METHOD M_SetSingleProp : ERRORID
VAR_INPUT
	refCmdData : REFERENCE TO  ST_CmdData;
END_VAR
IF nSpecPropIndex = refCmdData.aHeader[1] THEN
	IF refCmdData.n32Data[0] > 0 AND refCmdData.n32Data[0] <= cNoOfValves THEN
		nValveNrVac := DINT_TO_USINT(refCmdData.n32Data[0]);
	ELSE
		M_SetSingleProp := E_ErrorIdObjMgmt.ERRORID_InvalidValveNumber;
	END_IF	
ELSE
	M_SetSingleProp := SUPER^.M_SetSingleProp(refCmdData);
END_IF
END_METHOD

END_FUNCTION_BLOCK

// ---- Hardware/HuberUnistat/FB_UnistatControl.TcPOU
FUNCTION_BLOCK FB_UnistatControl
VAR_INPUT
	UnistatRef 		: REFERENCE TO FB_HwRefUnistat;
	nTempSetpoint 	: DINT;
	bTempControlOn	: BOOL;
	bExecute		: BOOL;
END_VAR
VAR_OUTPUT
	bBusy			: BOOL;
	bError			: BOOL;
	nErrorID		: ERRORID;
END_VAR
VAR
	fbSendCmd 		: FB_Unistat_SendCmd;
	nState			: UINT;
END_VAR

IF bExecute THEN
	IF NOT __ISVALIDREF(UnistatRef) THEN
		{warnig 'Implement proper ErrorID'}
		bError := TRUE;
		nErrorID := 333;
		RETURN;
	END_IF
	fbSendCmd.SerialPort REF= UnistatRef.P_SerialPort;
 	UnistatRef.P_bPolling := FALSE;
	
	IF nState = 0 THEN
		IF UnistatRef.P_eState = E_UnistatState.Error THEN
			RETURN;
		END_IF
		IF bTempControlOn THEN
			IF UnistatRef.P_eState = E_UnistatState.On THEN
				nState := 3;
			ELSE
				nState := 1;
			END_IF
		ELSE
			IF UnistatRef.P_eState = E_UnistatState.On THEN
				nState := 2;
			ELSE
				RETURN;
			END_IF
		END_IF
		bBusy := TRUE;
	END_IF
	
	CASE nState OF
		1:	//Ein
			fbSendCmd(bExecute:= TRUE, eCommand:= E_Unitstat_Command.Start_TempControl);
			IF NOT fbSendCmd.bBusy THEN
				fbSendCmd(bExecute:= FALSE);
				nState := 3;
			END_IF
		
		2:	//Aus
			fbSendCmd(bExecute:= TRUE, eCommand:= E_Unitstat_Command.Stop_TempControl);
			IF NOT fbSendCmd.bBusy THEN
				fbSendCmd(bExecute:= FALSE);
				bBusy := FALSE;
				nState := 80;
			END_IF
		
		3:	//Solltemperatur
			fbSendCmd(bExecute:= TRUE, eCommand:= E_Unitstat_Command.Set_TempSetPoint, nSendData := nTempSetPoint);
			IF NOT fbSendCmd.bBusy THEN
				fbSendCmd(bExecute:= FALSE);
				bBusy := FALSE;
				nState := 80;
			END_IF
	END_CASE
ELSE
	IF __ISVALIDREF(UnistatRef) THEN
		UnistatRef.P_bPolling := TRUE;
	END_IF
	nState := 0;
	bBusy := FALSE;
	bError := FALSE;
	nErrorID := 0;
END_IF

END_FUNCTION_BLOCK

// ---- Hardware/HuberUnistat/FB_HwRefUnistat.TcPOU
FUNCTION_BLOCK FB_HwRefUnistat
VAR_INPUT
END_VAR
VAR_OUTPUT
END_VAR
VAR
	SerialPort 	: REFERENCE TO FB_SerialComPort_Base;
	fbSendCmd 	: FB_Unistat_SendCmd;
	
	bPolling			: BOOL := TRUE;
	nCurrentTempIntern 	: DINT;
	nCurrentTempExtern 	: DINT;
	eState				: E_UnistatState;
	nState				: USINT;
	nStateNext			: USINT := 1;
END_VAR

IF NOT __ISVALIDREF(SerialPort) THEN
	RETURN;
END_IF
fbSendCmd.SerialPort REF= SerialPort;
IF NOT SerialPort.bIsWorking THEN
	RETURN;
END_IF

IF nState = 0 THEN
	IF bPolling THEN
		nState := nStateNext;
	END_IF
END_IF

CASE nState OF
	1:	//Status abrufen
		fbSendCmd(bExecute:= TRUE, eCommand:= E_Unitstat_Command.Get_Status);
		IF NOT fbSendCmd.bBusy THEN
			IF NOT fbSendCmd.bError THEN
				eState := fbSendCmd.nReceiveData;
			END_IF
			fbSendCmd(bExecute:= FALSE);
			nState := 0;
			nStateNext := 2;
		END_IF	

	2:	//Temp intern abrufen
		fbSendCmd(bExecute:= TRUE, eCommand:= E_Unitstat_Command.Get_TempActualIntern);
		IF NOT fbSendCmd.bBusy THEN
			IF fbSendCmd.bError THEN
				nCurrentTempIntern := 16#FFFF;
			ELSE
				nCurrentTempIntern := fbSendCmd.nReceiveData;
			END_IF
			fbSendCmd(bExecute:= FALSE);
			nState := 0;
			nStateNext := 3;
		END_IF
	3:	//Temp extern abrufen
		fbSendCmd(bExecute:= TRUE, eCommand:= E_Unitstat_Command.Get_TempActualExtern);
		IF NOT fbSendCmd.bBusy THEN
			IF fbSendCmd.bError THEN
				nCurrentTempExtern := 16#FFFF;
			ELSE
				IF fbSendCmd.nReceiveData = -1510 THEN
					nCurrentTempExtern := 16#FFFF;
				ELSE
					nCurrentTempExtern := fbSendCmd.nReceiveData;	
				END_IF
			END_IF
			fbSendCmd(bExecute:= FALSE);
			nState := 1;
			nStateNext := 1;
		END_IF
END_CASE

METHOD FB_init : BOOL
VAR_INPUT
	bInitRetains : BOOL; // if TRUE, the retain variables are initialized (warm start / cold start)
	bInCopyCode : BOOL;  // if TRUE, the instance afterwards gets moved into the copy code (online change)
	SerialPort 	: REFERENCE TO FB_SerialComPort_Base;
END_VAR
THIS^.SerialPort REF= SerialPort;
END_METHOD

PROPERTY P_bPolling : BOOL
GET
P_bPolling := bPolling;
END_GET
SET
bPolling := P_bPolling;
END_SET
END_PROPERTY

PROPERTY P_eState : E_UnistatState
GET
P_eState := eState;
END_GET
END_PROPERTY

PROPERTY P_nCurrentTempExtern : DINT
GET
P_nCurrentTempExtern := nCurrentTempExtern;
END_GET
END_PROPERTY

PROPERTY P_nCurrentTempIntern : DINT
GET
P_nCurrentTempIntern := nCurrentTempIntern;
END_GET
END_PROPERTY

PROPERTY P_SerialPort : REFERENCE TO FB_SerialComPort_Base
GET
P_SerialPort REF= SerialPort;
END_GET
END_PROPERTY

END_FUNCTION_BLOCK

// ---- Hardware/HuberUnistat/FB_Unistat_SendCmd.TcPOU
FUNCTION_BLOCK FB_Unistat_SendCmd
VAR_INPUT
	bExecute		: BOOL;	
	eCommand		: E_Unitstat_Command;
	nSendData		: DINT;
	SerialPort		: REFERENCE TO FB_SerialComPort_Base;	
END_VAR

VAR_OUTPUT
	bBusy			: BOOL;
	bError			: BOOL;
	nErrorId		: ERRORID; 		//RS232-Fehler oder vom Diluter zurückgegebener Fehler
	nReceiveData	: DINT;
END_VAR
VAR
	
	fbSendString	: Tc2_SerialCom.SendString;
	fbReceiveString	: Tc2_SerialCom.ReceiveString;
	bExpectReply	: BOOL;
	bExpectReal		: BOOL;
	rTemp			: REAL;
	sSendString		: STRING;
	sReceivedString	: STRING;
	sTemp			: STRING;
	
	nState			: USINT;
	bFlag			: BOOL := TRUE;
	nLenData		: USINT; //komplette Länge der Sende-oder Empfamgsdaten
	timeout			: TON;
END_VAR

IF bExecute THEN
	IF nState = 0 THEN
		IF NOT __ISVALIDREF(SerialPort) THEN
			bError := TRUE;
			RETURN;
		END_IF
		//Am Serial Port zu Senden registrieren
		//Die Registrierung sollte, wenn alles richtig programmiert wurde, immer klappen!
		IF NOT SerialPort.M_Register(THIS) THEN
			bError := TRUE;
			RETURN;
		ELSE
			nState := 1	;
		END_IF
		bBusy := TRUE;
	END_IF
	
	//Checken, ob an der Reihe (wird übersprungen, wenn "SerialPort.M_Register" TRUE zurückgibt
	IF nState = 1 THEN
		IF SerialPort.M_IsMyTurn(THIS) THEN
			nState := 2;
		END_IF
	END_IF
	
	//Ist für eine Zeit gesperrt und wird automatisch aufgehoben
	IF SerialPort.bIsLocked THEN
		RETURN;
	END_IF
	
	//Ist an der Reihe
	IF nState = 2 THEN
		//Kommunikationspuffer löschen (nicht der Hardware-Buffer)
		SerialPort.M_ClearTxComBuffer();
		SerialPort.M_ClearRxComBuffer();
		
		//# # # # # # # # # # # # # Sendestring zusammensetzen # # # # # # # # # # # # # # # # # # #
		CASE eCommand OF
			E_Unitstat_Command.Get_TempActualIntern:
				sSendString := 'IN_PV_00';
				bExpectReply := TRUE;
				bExpectReal := TRUE;
			E_Unitstat_Command.Get_TempActualExtern:
				sSendString := 'IN_PV_02';
				bExpectReply := TRUE;
				bExpectReal := TRUE;
			E_Unitstat_Command.Get_TempSetPoint:
				sSendString := 'IN_SP_00';
				bExpectReply := TRUE;
				bExpectReal := TRUE;
			E_Unitstat_Command.Get_Status:
				sSendString := 'STATUS';
				bExpectReply := TRUE;
			E_Unitstat_Command.Set_TempSetPoint:
				//Umwandlung von Ganzzahl 1/10tel°C in String als Gleitpunktzahl 
				rTemp := DINT_TO_REAL(nSendData) / 10.0;
				sSendString := CONCAT('OUT_SP_00 ', REAL_TO_STRING(rTemp));
			E_Unitstat_Command.Start_TempControl:
				sSendString := 'START';
			E_Unitstat_Command.Stop_TempControl:
				sSendString := 'STOP';
		ELSE
			bError := TRUE;
			RETURN;
		END_CASE
		
		//CR und LF anfügen
		sSendString := CONCAT(sSendString,'$R$N');
		nState := 3;	//weiter zu String senden
	END_IF
	
	CASE nState OF
		3:	//# # # # # # # # # # # # # Daten senden # # # # # # # # # # # # # # # # # # #
			IF bFlag XOR fbSendString.Busy THEN
				bFlag := FALSE;
				fbSendString(SendString:= sSendString, TXbuffer:= SerialPort.P_TxBuffer);
			END_IF
			
			IF NOT fbSendString.Busy THEN	//Sendung abgeschlossen
				IF fbSendString.Error > 0 THEN
					nErrorId := INT_TO_UINT(fbSendString.Error);
					bError := TRUE;
					bBusy := FALSE;
					nState := 99;
					RETURN;				
				ELSE
					IF bExpectReply THEN	//Antwort wird erwartet
						nState := 4;	//weiter zu Daten empfangen
					ELSE	//Antwort wird nicht erwartet -> Daten nicht abrufen
						//Hier muss SerialPort für 500ms blockiert werden (siehe Doku Unistat)
						SerialPort.M_LockForTime(T#500MS); 
						bBusy := FALSE;
						nState:= 80;
					END_IF
				END_IF
			END_IF
			
		4:	//# # # # # # # # # # # # # Daten empfangen # # # # # # # # # # # # # # # # # # #
			timeout(IN:= TRUE, PT:= T#500MS);
			IF timeout.Q THEN //Es wurden keine Daten mit entsprechendem Suffix empfangen -> Baustein resetten
				fbReceiveString(ReceivedString:= sReceivedString, RXbuffer:= SerialPort.P_RxBuffer, Reset:= TRUE);
				nErrorId := E_ErrorIdDiluter.ERRORID_ComTimeout;
				bError := TRUE;
				bBusy := FALSE;
				nState := 99;
			ELSE
				fbReceiveString(ReceivedString:= sReceivedString, Suffix:= '$R$N', RXbuffer:= SerialPort.P_RxBuffer, Reset:= FALSE);
				IF fbReceiveString.Error <> ComError_t.COMERROR_NOERROR THEN
					fbReceiveString(ReceivedString:= sReceivedString, RXbuffer:= SerialPort.P_RxBuffer, Reset:= TRUE);
					bError := TRUE;
					bBusy := FALSE;
					nErrorId := INT_TO_UINT(fbReceiveString.Error);
					nState := 99;
					RETURN;
				END_IF
				
				IF fbReceiveString.StringReceived THEN
					IF bExpectReal THEN
						nReceiveData := REAL_TO_DINT(STRING_TO_REAL(sReceivedString) * 10.0);	
					ELSE
						nReceiveData := STRING_TO_DINT(sReceivedString);
					END_IF
					SerialPort.M_LockForTime(T#500MS);
					bBusy := FALSE;
					nState := 80;
				END_IF
			END_IF
	END_CASE
ELSE
	IF __ISVALIDREF(SerialPort) AND_THEN SerialPort.M_IsMyTurn(THIS) THEN
		SerialPort.M_Release(THIS);
	END_IF
	bBusy := FALSE;
	bError := FALSE;
	bExpectReply := FALSE;
	bExpectReal := FALSE;
	bFlag := TRUE;
	nErrorId := 0;
	nState := 0;
	nReceiveData := 0;
	timeout(IN:= FALSE);
END_IF

END_FUNCTION_BLOCK

// ---- Objects/Targets/Active/FB_LiquidReserve.TcPOU
FUNCTION_BLOCK FB_LiquidReserve EXTENDS FB_ActiveTarget
VAR
	aLevelSensor		AT %I* : ARRAY[1..cMaxSlots] OF BOOL; 		
	
	//Spec-Properties

	nNoOfSlots			: USINT;
	nNoOfSpecPoints		: USINT;
	nNoOfWasteChannels	: USINT;
	nNoOfLiquidChannels	: USINT;
	
	aSlots				: ARRAY[1..cMaxSlots] OF FB_PieceSlot(pOwner:= This);
	aSpecPoints			: ARRAY[1..cMaxSpecPoints] OF ST_3DPoint;
	aWasteChannels		: ARRAY[1..cMaxWasteChannels] OF ST_WasteChannel;
	aLiquidChannels		: ARRAY[1..cMaxLiquidChannels] OF ST_LiquidChannel;
	//aFbGearPump			: ARRAY[1..cMaxLiquidChannels] OF FB_GearPump(stCANInterfaceBuffer := CANInterfaceCom.stCanInterfaceBuffer);
	nPumpNr				: USINT;

	//Variablen allgemeine Statemachine
	
	
	//****************************************Aktionvariablen****************************************************
	
	nChannelCnt			: USINT;	//allg.Zählvariable für For Next-Schleifen
	
	//Action: "FillLiquid"
	bFillLiquid				: BOOL;

	//Action: "EmptyLiquid"
	bEmptyLiquid			: BOOL;

	nStateA_FillEmptyLiquid		: USINT;
	aFillEmptyLiquid			: ARRAY[1..cMaxLiquidChannels] OF BOOL;
	aSubStateA_FillEmptyLiquid 	: ARRAY[1..cMaxLiquidChannels] OF USINT;
	
	nFillEmptyChannel			: USINT;
	aFillEmptyQuantity			: ARRAY[1..cMaxLiquidChannels] OF DINT;
	aFillEmptyFlow				: ARRAY[1..cMaxLiquidChannels] OF DINT;
	
	//Action: EmptyWaste
	bEmptyWaste				: BOOL;
	nStateA_EmptyWaste		: USINT;
	nEmptyWasteChannel		: USINT;
	tEmptyTime				: TIME;
	tmrEmptyWaste			: TON;

END_VAR

VAR CONSTANT
	cMaxSlots 			: USINT := 6;
	cMaxSpecPoints		: USINT := 2;
	cMaxLiquidChannels 	: USINT := 4;
	cMaxWasteChannels 	: USINT := 2;
END_VAR

IF bInitFB THEN
	bInitFB := FALSE;
	F_CreateLinkedListHnd( ADR( aNodes ), SIZEOF( aNodes ), hList );
	//Fehlerstruktur vorausfüllen
	stError.ObjectId := nObjectID;
	stError.HardwareGrp := E_HardwareGrp.Nothing;
	stError.POU := E_POU.POU_FB_LiquidReserve;
	//Pumpennummer zu den Instanzen von FB_GearPump zuordnen
	
END_IF

FOR nPumpNr := 1 TO cMaxLiquidChannels BY 1 DO
	//aFbGearPump[nPumpNr](stTMCMBuffer := stTMCMBuffer, nPumpNr := nPumpNr);
	//aFbGearPump[nPumpNr](nPumpNr:=nPumpNr);
END_FOR

CASE eCurrentState OF
	E_MachineState.MACHINESTATE_Active:
		//BasicActions ausführen
		IF bInit THEN	//Initialisieren
			A_Init();
			IF nStateA_Init >= 80 THEN
				IF nStateA_Init >= 99 THEN
					fbErrorList.M_Add(stError);	//Error in Error-Liste eintragen
					bError := TRUE;	
				END_IF
				bInit := FALSE;
				nStateA_Init := 0;
				M_RemoveListEntry(nSearchValue:= E_Action.ACTION_Init);
			END_IF
		END_IF
		
		IF bFillLiquid THEN
			A_FillLiquid();
			IF nStateA_FillEmptyLiquid >= 80 THEN
				IF nStateA_FillEmptyLiquid >= 99 THEN
					fbErrorList.M_Add(stError);	//Error in Error-Liste eintragen
					bError := TRUE;
				END_IF
				bFillLiquid := FALSE;
				nStateA_FillEmptyLiquid := 0;
				M_RemoveListEntry(nSearchValue:= E_Action.ACTION_FillLiquid);
			END_IF
		END_IF
		
		IF bEmptyLiquid THEN
			A_EmptyLiquid();
			IF nStateA_FillEmptyLiquid >= 80 THEN
				IF nStateA_FillEmptyLiquid >= 99 THEN
					fbErrorList.M_Add(stError);	//Error in Error-Liste eintragen
					bError := TRUE;
				END_IF
				bEmptyLiquid := FALSE;
				nStateA_FillEmptyLiquid := 0;
				M_RemoveListEntry(nSearchValue:= E_Action.ACTION_EmptyLiquid);
			END_IF
		END_IF
		
		IF bEmptyWaste THEN
			A_EmptyWaste();
			IF nStateA_EmptyWaste >= 80 THEN
				IF nStateA_EmptyWaste >= 99 THEN
					fbErrorList.M_Add(stError);	//Error in Error-Liste eintragen
					bError := TRUE;
				END_IF
				bEmptyWaste := FALSE;
				nStateA_EmptyWaste := 0;
				M_RemoveListEntry(nSearchValue:= E_Action.ACTION_EmptyWaste);
			END_IF
		END_IF
		
		IF bStop THEN
			A_Stop();
			IF nStateA_Stop >= 80 THEN
				IF nStateA_Stop >= 99 THEN
					fbErrorList.M_Add(stError);	//Error in Error-Liste eintragen
					bError := TRUE;
				END_IF
				bStop := FALSE;
				nStateA_Stop := 0;
				bStop := FALSE;
				M_RemoveListEntry(nSearchValue:= E_Action.ACTION_Stop);
			END_IF							
		END_IF		
		
		IF hList.nCount = 0 THEN
			eCurrentState := E_MachineState.MACHINESTATE_Ready;
		END_IF

		IF bError  THEN
			eCurrentState := E_MachineState.MACHINESTATE_Error;
		END_IF

	E_MachineState.MACHINESTATE_Reset:
		A_Reset();
		IF nStateA_Reset = 80 THEN
			nStateA_Init := 0;
			nStateA_Stop := 0;
			nStateA_Reset := 0;
			bBusy := FALSE;
			bError := FALSE;
			bStopAllOnError := FALSE;
			fbList.A_Reset( hList := hList);
			nErrorId := 0;
			stError.Cmd := 0;
			stError.ErrorId := 0;
			eCurrentState := E_MachineState.MACHINESTATE_Idle;
		ELSIF
			nStateA_Reset = 99 THEN
			fbErrorList.M_Add(stError);
			nStateA_Reset := 0;
			bBusy := FALSE;
			bError := TRUE;
			eCurrentState := E_MachineState.MACHINESTATE_Error;			
		END_IF
	
	E_MachineState.MACHINESTATE_Ready:
		bBusy := FALSE;
		eCurrentState := E_MachineState.MACHINESTATE_Idle;
	
	E_MachineState.MACHINESTATE_Error:
		bBusy := FALSE;
END_CASE

//Prozessdaten aktualisieren
stProcessData.nObjId := nObjectID;
stProcessData.n32Data[0] := BOOL_TO_DINT(bIsInit);
stProcessData.n32Data[1] := eCurrentState;
stProcessData.n32Data[2] := stError.ErrorId;

aObjProcData[nNotifyId] := stProcessData;

ACTION A_EmptyLiquid:
IF nStateA_FillEmptyLiquid = 0 THEN
	//Die einzelnen Channels durchlaufen
	//Die einzelnen Channels haben ihre eigene Statemachine
	//In diesem State werden auch geändert Werte angenommen
	nStateA_FillEmptyLiquid := 80;
	FOR nChannelCnt := 1 TO cMaxLiquidChannels BY 1 DO
		CASE aSubStateA_FillEmptyLiquid[nChannelCnt] OF
			0:
				IF aFillEmptyLiquid[nChannelCnt] THEN
					aFillEmptyLiquid[nChannelCnt] := FALSE;
					nStateA_FillEmptyLiquid := 0;
					aLiquidChannels[nChannelCnt].pGearPump^.M_PumpQuantity(aFillEmptyQuantity[nChannelCnt],aFillEmptyFlow[nChannelCnt]);
					aSubStateA_FillEmptyLiquid[nChannelCnt] := 1;
				END_IF
			1:	//Warten bis fertig
				IF aLiquidChannels[nChannelCnt].pGearPump^.bBusy THEN
					nStateA_FillEmptyLiquid := 0;
				ELSE
					aSubStateA_FillEmptyLiquid[nChannelCnt] := 0;
				END_IF
		END_CASE
	END_FOR
ELSIF nStateA_FillEmptyLiquid = 70 THEN
	nStateA_FillEmptyLiquid := 80;
	FOR nChannelCnt := 1 TO cMaxLiquidChannels BY 1 DO
		aLiquidChannels[nChannelCnt].pGearPump^.M_Stop();
		IF aLiquidChannels[nChannelCnt].pGearPump^.bBusy THEN
			nStateA_FillEmptyLiquid := 70;
		END_IF
	END_FOR
END_IF
END_ACTION

ACTION A_EmptyWaste:
IF nStateA_EmptyWaste = 0 THEN
	FOR nChannelCnt := 1 TO cMaxWasteChannels BY 1 DO
		aPumps[aWasteChannels[nChannelCnt].nPumpNr].M_Off();
		IF 	nEmptyWasteChannel = 0 THEN //Alle leeren
			aPumps[aWasteChannels[nChannelCnt].nPumpNr].M_On();
		ELSIF nEmptyWasteChannel = nChannelCnt THEN
			aPumps[aWasteChannels[nChannelCnt].nPumpNr].M_On();
		END_IF
	END_FOR
	tmrEmptyWaste(IN:= TRUE, PT:= tEmptyTime);
	IF tmrEmptyWaste.Q THEN
		FOR nChannelCnt := 1 TO cMaxWasteChannels BY 1 DO
			aPumps[aWasteChannels[nChannelCnt].nPumpNr].M_Off();
		END_FOR
		nStateA_EmptyWaste := 80;		
	END_IF
ELSIF nStateA_EmptyWaste = 70 THEN
	nStateA_EmptyWaste := 80;
	FOR nChannelCnt := 1 TO cMaxWasteChannels BY 1 DO
		aPumps[aWasteChannels[nChannelCnt].nPumpNr].M_Off();
	END_FOR
END_IF
END_ACTION

ACTION A_FillLiquid:
FOR nChannelCnt := 1 TO cMaxWasteChannels BY 1 DO
	aPumps[aWasteChannels[nChannelCnt].nPumpNr].M_Off();
END_FOR

IF nStateA_FillEmptyLiquid = 0 THEN
	//Die einzelnen Channels durchlaufen
	//Die einzelnen Channels haben ihre eigene Statemachine
	//In diesem State werden auch geändert Werte angenommen
	nStateA_FillEmptyLiquid := 80;
	FOR nChannelCnt := 1 TO cMaxLiquidChannels BY 1 DO
		//Sensoren der Bottles überwachen
		IF aFillEmptyFlow[nChannelCnt] > 0 THEN
			IF aLiquidChannels[nChannelCnt].nBottleNr > 0 THEN
				IF NOT aSensSysLiquidBottle[aLiquidChannels[nChannelCnt].nBottleNr] THEN //Leer
					stError.ErrorId := E_ErrorIdCmd.ERRORID_LiquidBottleEmpty;
					nStateA_FillEmptyLiquid := 99;
				END_IF
			END_IF
			IF aWasteChannels[aLiquidChannels[nChannelCnt].nWasteCh].nBottleNr > 0 THEN
				IF NOT aSensWasteBottle[aWasteChannels[aLiquidChannels[nChannelCnt].nWasteCh].nBottleNr] THEN
					stError.ErrorId := E_ErrorIdCmd.ERRORID_WasteBottleFull;
					nStateA_FillEmptyLiquid := 99;
				END_IF
			END_IF
		END_IF
		IF nStateA_FillEmptyLiquid < 99 THEN
			CASE aSubStateA_FillEmptyLiquid[nChannelCnt] OF
				0:
					IF aFillEmptyLiquid[nChannelCnt] THEN
						aFillEmptyLiquid[nChannelCnt] := FALSE;
						//zugeordnete WastePump einschalten
						//Befehl absenden
						//Wenn eine Menge vorgegeben, dann M_PumpQuantity, sonse M_PumpConst
						nStateA_FillEmptyLiquid := 0;
						IF aFillEmptyQuantity[nChannelCnt] = 0 THEN
							aLiquidChannels[nChannelCnt].pGearPump^.M_PumpConst(aFillEmptyFlow[nFillEmptyChannel]);
						ELSE
							aLiquidChannels[nChannelCnt].pGearPump^.M_PumpQuantity(aFillEmptyQuantity[nChannelCnt],aFillEmptyFlow[nChannelCnt]);
						END_IF
						aSubStateA_FillEmptyLiquid[nChannelCnt] := 1;
					END_IF
				1:
					//Wartet bis fertig, nimmt aber auch neuen Befehl an
					//Wenn Füllstandssensor, dann auch abschalten
					IF aFillEmptyLiquid[nChannelCnt] THEN
						aSubStateA_FillEmptyLiquid[nChannelCnt] := 0;
						nStateA_FillEmptyLiquid := 0;
					ELSE
						IF NOT aLiquidChannels[nChannelCnt].pGearPump^.bBusy THEN
							aSubStateA_FillEmptyLiquid[nChannelCnt] := 0;
							aFillEmptyFlow[nChannelCnt] := 0;
						ELSE
							IF NOT aLevelSensor[nChannelCnt] THEN
								IF aFillEmptyQuantity[nChannelCnt] = 0 THEN
									aLiquidChannels[nChannelCnt].pGearPump^.M_Stop();
									aFillEmptyFlow[nChannelCnt] := 0;
								END_IF
							END_IF
							nStateA_FillEmptyLiquid := 0;
						END_IF
					END_IF
			END_CASE
			IF aLiquidChannels[nChannelCnt].pGearPump^.bBusy THEN
				aPumps[aWasteChannels[aLiquidChannels[nChannelCnt].nWasteCh].nPumpNr].M_On();
			END_IF
		END_IF
	END_FOR
ELSIF nStateA_FillEmptyLiquid = 70 THEN
	//WastePumps ausschalten
	FOR nChannelCnt := 1 TO cMaxWasteChannels BY 1 DO
		aPumps[aWasteChannels[nChannelCnt].nPumpNr].M_Off();
	END_FOR
	
	nStateA_FillEmptyLiquid := 80;
	FOR nChannelCnt := 1 TO cMaxLiquidChannels BY 1 DO
		aLiquidChannels[nChannelCnt].pGearPump^.M_Stop();
		IF aLiquidChannels[nChannelCnt].pGearPump^.bBusy THEN
			nStateA_FillEmptyLiquid := 70;
		END_IF
	END_FOR
END_IF

//Errorhandling
IF nStateA_FillEmptyLiquid = 99 THEN
	//Alle Pumpen ausschalten
	FOR nChannelCnt := 1 TO cMaxLiquidChannels BY 1 DO
		aLiquidChannels[nChannelCnt].pGearPump^.M_Stop();
		aFillEmptyFlow[nChannelCnt] := 0;
	END_FOR
	
	FOR nChannelCnt := 1 TO cMaxWasteChannels BY 1 DO
		aPumps[aWasteChannels[nChannelCnt].nPumpNr].M_Off();
	END_FOR

	stError.Cmd := E_Action.ACTION_FillLiquid;
	stError.POUAction := E_POUACT.POUACT_A_FillLiquid;
	fbErrorList.M_Add(stError);
END_IF
END_ACTION

ACTION A_Init:
nStateA_Init := 80;
END_ACTION

ACTION A_Reset:
CASE nStateA_Reset OF
	0:
		nStateA_Reset := 80;
END_CASE
END_ACTION

ACTION A_Stop:
CASE nStateA_Stop OF
	0:	//Fehlerstruktur vorausfüllen
		stError.Cmd := E_Action.ACTION_Stop;
		IF bInit THEN
			nStateA_Init := 70;	
		END_IF
		
		nStateA_Stop := 1;
	
	1:	//Warten bis alle Actions außer Stop abgebrochen sind
		IF hList.nCount = 1 THEN	//nur der Eintrag von Stop
			nStateA_Stop := 80;
		END_IF
END_CASE
END_ACTION

METHOD FB_init : BOOL
VAR_INPUT
	bInitRetains : BOOL; // if TRUE, the retain variables are initialized (warm start / cold start)
	bInCopyCode : BOOL;  // if TRUE, the instance afterwards gets moved into the copy code (online change)
END_VAR
eObjectType := E_ObjectType.OBJECTTYPE_LiquidReserve;
eObjectGroup := E_ObjectGroup.OBJECTGROUP_Target OR E_ObjectGroup.OBJECTGROUP_Device;
END_METHOD

METHOD M_ApplyPos : ERRORID
VAR_INPUT
	eTargetRef 		: E_TargetRef;
	nPointSlotNr	: UINT;
	stPos 			: ST_3DPoint;
	bXPos			: BOOL;
	bYPos			: BOOL;
	bZPos			: BOOL;	
END_VAR

VAR
	stAbsPos		: ST_3DPoint;
END_VAR
stAbsPos := P_stAbsPosLB;
IF eTargetRef = E_TargetRef.TARGETREF_SpecPoint THEN
	IF nPointSlotNr > 0 AND nPointSlotNr <= nNoOfSpecPoints THEN
		IF bXPos THEN
			aSpecPoints[nPointSlotNr].X := stPos.X - stAbsPos.X;	
		END_IF
		IF bYPos THEN
			aSpecPoints[nPointSlotNr].Y := stPos.Y - stAbsPos.Y;	
		END_IF
		IF bZPos THEN
			aSpecPoints[nPointSlotNr].Z := stPos.Z - stAbsPos.Z;	
		END_IF
	ELSE
		M_ApplyPos := E_ErrorIdCmd.ERRORID_InvalidTargetPointNr;
	END_IF
ELSIF eTargetRef = E_TargetRef.TARGETREF_Slot THEN
	IF nPointSlotNr > 0 AND nPointSlotNr <= nNoOfSlots THEN
		IF bXPos THEN
			aSlots[nPointSlotNr].P_rRelPosX := stPos.X - stAbsPos.X;	
		END_IF
		IF bYPos THEN
			aSlots[nPointSlotNr].P_rRelPosY := stPos.Y - stAbsPos.Y;	
		END_IF
		IF bZPos THEN
			aSlots[nPointSlotNr].P_rRelPosZ := stPos.Z - stAbsPos.Z;	
		END_IF
	ELSE
		M_ApplyPos := E_ErrorIdCmd.ERRORID_InvalidTargetPointNr;
	END_IF
ELSE
	M_ApplyPos := SUPER^.M_ApplyPos(eTargetRef, nPointSlotNr, stPos,bXPos, bYPos, bZPos);
END_IF
END_METHOD

METHOD M_CancelAction
VAR_INPUT
	eAction : E_Action;
END_VAR
CASE eAction OF
	E_Action.ACTION_FillLiquid:
		IF bFillLiquid AND nStateA_FillEmptyLiquid < 70 THEN
			nStateA_FillEmptyLiquid := 70;
		END_IF	
	E_Action.ACTION_EmptyLiquid:
		IF bEmptyLiquid AND nStateA_FillEmptyLiquid < 70 THEN
			nStateA_FillEmptyLiquid := 70;
		END_IF
	E_Action.ACTION_EmptyWaste:
		IF bEmptyWaste AND nStateA_EmptyWaste < 70 THEN
			nStateA_EmptyWaste := 70;
		END_IF
END_CASE
END_METHOD

METHOD M_CheckBottles : ERRORID
VAR_INPUT
END_VAR
//Systemliquidbottle OK?
(*IF nSysLiquidBottle > 0 THEN
	IF NOT aSensSysLiquidBottle[nSysLiquidBottle] THEN //Leer
		M_GetBottleState := E_ErrorIdCmd.ERRORID_LiquidBottleEmpty;
		RETURN;
	END_IF
END_IF
//Wastebottle OK?
IF nWasteBottle > 0 THEN
	IF NOT aSensWasteBottle[nWasteBottle] THEN //Voll
		M_GetBottleState := E_ErrorIdCmd.ERRORID_WasteBottleFull;
		RETURN;
	END_IF
END_IF*)
END_METHOD

METHOD M_CheckForAction : BOOL
VAR_INPUT
	refActionData : REFERENCE TO ST_ActionData;
END_VAR
IF refActionData.eAction = E_Action.ACTION_TeachTarget THEN
	IF DINT_TO_UINT(refActionData.aParams[1]) = E_TargetRef.TARGETREF_SpecPoint AND (refActionData.aParams[2] = 1 AND refActionData.aParams[2] = 2) THEN
		M_CheckForAction := TRUE;
	END_IF
END_IF
END_METHOD

METHOD M_CheckProcDataType : BOOL
VAR_INPUT
	eProcDataType : E_ProcDataType;
END_VAR
END_METHOD

METHOD M_ExeAction : ERRORID
VAR_INPUT
	refActionData : REFERENCE TO ST_ActionData;	
END_VAR
IF refActionData.eAction = E_Action.ACTION_Init THEN
	bIsInit := TRUE;
	RETURN;
ELSIF refActionData.eAction = E_Action.ACTION_FillLiquid THEN
	IF bEmptyLiquid THEN
		M_ExeAction := E_ErrorIdCmd.ERRORID_BasicActionActive;
	END_IF

	nFillEmptyChannel := DINT_TO_USINT(refActionData.aParams[3]);
	IF nFillEmptyChannel > cMaxLiquidChannels THEN
		M_ExeAction := E_ErrorIdCmd.ERRORID_InvalidLiquidChannel;
		RETURN;
	END_IF

	aFillEmptyQuantity[nFillEmptyChannel] := refActionData.aParams[1];
	aFillEmptyFlow[nFillEmptyChannel] := refActionData.aParams[2];
	aFillEmptyLiquid[nFillEmptyChannel] := TRUE;
	
	IF NOT bFillLiquid THEN
		fbList.A_AddHeadValue(hList := hList, putValue:= E_Action.ACTION_FillLiquid);
		bFillLiquid := TRUE;
	END_IF
	
ELSIF refActionData.eAction = E_Action.ACTION_EmptyLiquid THEN
	IF bFillLiquid THEN
		M_ExeAction := E_ErrorIdCmd.ERRORID_BasicActionActive;
	END_IF
	
	nFillEmptyChannel := DINT_TO_USINT(refActionData.aParams[3]);
	IF nFillEmptyChannel > cMaxLiquidChannels THEN
		M_ExeAction := E_ErrorIdCmd.ERRORID_InvalidLiquidChannel;
		RETURN;
	END_IF
	
	aFillEmptyQuantity[nFillEmptyChannel] := refActionData.aParams[1] * -1;
	aFillEmptyFlow[nFillEmptyChannel] := refActionData.aParams[2];
	aFillEmptyLiquid[nFillEmptyChannel] := TRUE;
	
	IF NOT bEmptyLiquid THEN
		fbList.A_AddHeadValue(hList := hList, putValue:= E_Action.ACTION_EmptyLiquid);
		bEmptyLiquid := TRUE;
	END_IF
ELSIF refActionData.eAction = E_Action.ACTION_EmptyWaste THEN
	nEmptyWasteChannel := DINT_TO_USINT(refActionData.aParams[1]);
	IF nEmptyWasteChannel >= 0 AND  nEmptyWasteChannel <= cMaxWasteChannels THEN
		tEmptyTime := DINT_TO_TIME(refActionData.aParams[2]);
		tmrEmptyWaste(IN:= FALSE);
		IF NOT bEmptyWaste THEN
			fbList.A_AddHeadValue(hList := hList, putValue:= E_Action.ACTION_EmptyWaste);
			bEmptyWaste := TRUE;
		END_IF	
	ELSE
		M_ExeAction := E_ErrorIdCmd.ERRORID_InvalidWasteChannel;
		RETURN;		
	END_IF
ELSIF refActionData.eAction = E_Action.ACTION_Stop THEN
	;
ELSE
	M_ExeAction := E_ErrorIdCmd.ERRORID_InvalidAction;
	RETURN;
END_IF
bBusy := TRUE;
eCurrentState:= E_MachineState.MACHINESTATE_Active;
END_METHOD

METHOD M_GetAbsPos : ST_3DPoint
VAR_INPUT
	pChildPos	: POINTER TO ST_3DPoint;
	eTargetRef 	: E_TargetRef;
	nParam1		: UINT;
 	nParam2		: UINT;
	nParam3		: USINT;
	nParam4		: USINT;
	nZLevel		: USINT;
END_VAR
VAR_OUTPUT
	nErrorId 	: ERRORID;
	lrAngle		: LREAL;
END_VAR
VAR
	stLocPosLB : ST_3DPoint;
END_VAR
IF eTargetRef = E_TargetRef.TARGETREF_SpecPoint THEN
	IF nParam1 >= 1 AND nParam1 <= nNoOfSpecPoints THEN
		stLocPosLB := P_stRelPosLB;
		stLocPosLB := F_Add3DPoints(stLocPosLB,aSpecPoints[nParam1]);
		M_GetAbsPos := pParentTarget^.M_GetAbsPos(pChildPos := ADR(stLocPosLB), eTargetRef:= E_TargetRef.TARGETREF_LeftBottom,
													nParam1:= 0,
													nParam2:= 0, nParam3:= 0,nParam4:= 0, nZLevel:= 0,
													lrAngle => lrAngle, nErrorId=> nErrorId);		
	ELSE
		nErrorId := E_ErrorIdCmd.ERRORID_InvalidTargetPointNr;
	END_IF
	
ELSIF eTargetRef = E_TargetRef.TARGETREF_Slot THEN
	IF nParam1 >= 1 AND nParam1 <= nNoOfSlots THEN
		stLocPosLB := P_stRelPosLB;
		stLocPosLB := F_Add3DPoints(stLocPosLB,aSlots[nParam1].P_stRelPos);
		M_GetAbsPos := pParentTarget^.M_GetAbsPos(pChildPos := ADR(stLocPosLB), eTargetRef:= E_TargetRef.TARGETREF_LeftBottom,
													nParam1:= 0,
													nParam2:= 0, nParam3:= 0, nParam4:= 0, nZLevel:= 0,
													lrAngle => lrAngle, nErrorId=> nErrorId);			
	ELSE
		nErrorId := E_ErrorIdCmd.ERRORID_InvalidTargetPointNr;
	END_IF
ELSE
	M_GetAbsPos := SUPER^.M_GetAbsPos(pChildPos := pChildPos, eTargetRef:= eTargetRef,
													nParam1:= nParam1,
													nParam2:= nParam2, nParam3:= nParam3, nParam4:= 0, nZLevel:= nZLevel,
													lrAngle => lrAngle, nErrorId=> nErrorId);		
END_IF
END_METHOD

METHOD M_GetActionBusy : BOOL
VAR_INPUT
	eAction : E_Action;
END_VAR
IF eAction = E_Action.ACTION_FillLiquid THEN
	M_GetActionBusy := bFillLiquid;
ELSIF eAction = E_Action.ACTION_EmptyLiquid THEN
	M_GetActionBusy := bEmptyLiquid;
ELSIF eAction = E_Action.ACTION_EmptyWaste THEN
	M_GetActionBusy := bEmptyWaste;
END_IF
END_METHOD

METHOD M_GetAllProps : ERRORID
VAR_INPUT
	refCmdData : REFERENCE TO  ST_CmdData;
END_VAR

VAR
	i 		: USINT;
END_VAR
SUPER^.M_GetAllProps(refCmdData); 

//Slots
nCurrentPropIndex := nCurrentPropIndex + 1;
refCmdData.n32Data[nCurrentPropIndex] := nNoOfSlots;
FOR i := 1 TO nNoOfSlots BY 1 DO
	nCurrentPropIndex := nCurrentPropIndex + 1;
	refCmdData.n32Data[nCurrentPropIndex] := aSlots[i].nNr;
	nCurrentPropIndex := nCurrentPropIndex + 1;
	refCmdData.n32Data[nCurrentPropIndex] := REAL_TO_DINT(aSlots[i].stRelPos.X);
	nCurrentPropIndex := nCurrentPropIndex + 1;
	refCmdData.n32Data[nCurrentPropIndex] := REAL_TO_DINT(aSlots[i].stRelPos.Y);
	nCurrentPropIndex := nCurrentPropIndex + 1;
	refCmdData.n32Data[nCurrentPropIndex] := REAL_TO_DINT(aSlots[i].stRelPos.Z);
	nCurrentPropIndex := nCurrentPropIndex + 1;
	refCmdData.n32Data[nCurrentPropIndex] := REAL_TO_DINT(aSlots[i].rDepth);
END_FOR

//SpecPoints
nCurrentPropIndex := nCurrentPropIndex + 1;
refCmdData.n32Data[nCurrentPropIndex] := nNoOfSpecPoints;
FOR i := 1 TO nNoOfSpecPoints BY 1 DO
	nCurrentPropIndex := nCurrentPropIndex + 1;
	refCmdData.n32Data[nCurrentPropIndex] := REAL_TO_DINT(aSpecPoints[i].X);
	nCurrentPropIndex := nCurrentPropIndex + 1;
	refCmdData.n32Data[nCurrentPropIndex] := REAL_TO_DINT(aSpecPoints[i].Y);
	nCurrentPropIndex := nCurrentPropIndex + 1;
	refCmdData.n32Data[nCurrentPropIndex] := REAL_TO_DINT(aSpecPoints[i].Z);
END_FOR

//WasteChannles
nCurrentPropIndex := nCurrentPropIndex + 1;
refCmdData.n32Data[nCurrentPropIndex] := nNoOfWasteChannels;
FOR i := 1 TO nNoOfWasteChannels BY 1 DO
	nCurrentPropIndex := nCurrentPropIndex + 1;
	refCmdData.n32Data[nCurrentPropIndex] := aWasteChannels[i].nNr;
	nCurrentPropIndex := nCurrentPropIndex + 1;
	refCmdData.n32Data[nCurrentPropIndex] := aWasteChannels[i].nSpecPointNr;
	nCurrentPropIndex := nCurrentPropIndex + 1;
	refCmdData.n32Data[nCurrentPropIndex] := aWasteChannels[i].nPumpNr;
	nCurrentPropIndex := nCurrentPropIndex + 1;
	refCmdData.n32Data[nCurrentPropIndex] := aWasteChannels[i].nBottleNr;
END_FOR

//LiquidChannels
nCurrentPropIndex := nCurrentPropIndex + 1;
refCmdData.n32Data[nCurrentPropIndex] := nNoOfLiquidChannels;
FOR i := 1 TO nNoOfLiquidChannels BY 1 DO
	nCurrentPropIndex := nCurrentPropIndex + 1;
	refCmdData.n32Data[nCurrentPropIndex] := aLiquidChannels[i].nNr;
	nCurrentPropIndex := nCurrentPropIndex + 1;
	refCmdData.n32Data[nCurrentPropIndex] := aLiquidChannels[i].nSlotNr;
	nCurrentPropIndex := nCurrentPropIndex + 1;
	refCmdData.n32Data[nCurrentPropIndex] := aLiquidChannels[i].nWasteCh;
	nCurrentPropIndex := nCurrentPropIndex + 1;
	refCmdData.n32Data[nCurrentPropIndex] := aLiquidChannels[i].nBottleNr;
END_FOR
END_METHOD

METHOD M_GetProcData : DINT
VAR_INPUT
	eProcDataType : E_ProcDataType;
END_VAR
END_METHOD

METHOD M_RemoveListEntry : BOOL
VAR_INPUT
	nSearchValue	: E_Action;
END_VAR
getPosPtr := 0;(* start from first node element *)
fbList.A_FindNext( hList := hList, putPosPtr := getPosPtr, putValue := nSearchValue, getValue=>getValue, getPosPtr=>getPosPtr );
IF fbList.bOk THEN	//Eintrag wurde gefunden
	fbList.A_RemoveValueAtPosPtr(hList:= hList,	putPosPtr:= getPosPtr);
	IF fbList.bOk THEN
		M_RemoveListEntry := TRUE;
	END_IF
END_IF
END_METHOD

METHOD M_Reset
bError := FALSE;
bBusy := FALSE;
eCurrentState := E_MachineState.MACHINESTATE_Idle;
END_METHOD

METHOD M_SetAllProps : ERRORID
VAR_INPUT
	refCmdData : REFERENCE TO  ST_CmdData;
END_VAR

VAR
	i 		: USINT;
END_VAR
M_SetAllProps := SUPER^.M_SetAllProps(refCmdData);

IF M_SetAllProps > 0 THEN	//Error beim setzen der Base-Parameter
	RETURN;
END_IF

//Slots
nCurrentPropIndex := nCurrentPropIndex + 1;
nSpecPropIndex := nCurrentPropIndex;
IF refCmdData.n32Data[nCurrentPropIndex] >= 1 AND refCmdData.n32Data[nCurrentPropIndex] <= cMaxSlots THEN
	nNoOfSlots := DINT_TO_USINT(refCmdData.n32Data[nCurrentPropIndex]);
ELSE
	M_SetAllProps := E_ErrorIdObjMgmt.ERRORID_InvalidNoOfSlots;
	RETURN;
END_IF

FOR i:= 1 TO nNoOfSlots BY 1 DO
	nCurrentPropIndex := nCurrentPropIndex + 1;
	aSlots[i].P_nNr := DINT_TO_UINT(refCmdData.n32Data[nCurrentPropIndex]);
	nCurrentPropIndex := nCurrentPropIndex + 1;
	aSlots[i].P_rRelPosX := DINT_TO_REAL(refCmdData.n32Data[nCurrentPropIndex]);
	nCurrentPropIndex := nCurrentPropIndex + 1;
	aSlots[i].P_rRelPosY := DINT_TO_REAL(refCmdData.n32Data[nCurrentPropIndex]);
	nCurrentPropIndex := nCurrentPropIndex + 1;
	aSlots[i].P_rRelPosZ := DINT_TO_REAL(refCmdData.n32Data[nCurrentPropIndex ]);
	nCurrentPropIndex := nCurrentPropIndex + 1;
	aSlots[i].P_rDepth := DINT_TO_REAL(refCmdData.n32Data[nCurrentPropIndex]);
	aLiquidChannels[i].pGearPump := ADR(aFbGearPumps[i]);
END_FOR

//SpecPoints
nCurrentPropIndex := nCurrentPropIndex + 1;
IF refCmdData.n32Data[nCurrentPropIndex] >= 1 AND refCmdData.n32Data[nCurrentPropIndex] <= cMaxSpecPoints THEN
	nNoOfSpecPoints := DINT_TO_USINT(refCmdData.n32Data[nCurrentPropIndex]);
ELSE
	M_SetAllProps := E_ErrorIdObjMgmt.ERRORID_InvalidNoOfSpecPoints;
	RETURN;	
END_IF

//SpecPoints  parametrieren
FOR i:= 1 TO nNoOfSpecPoints BY 1 DO
	nCurrentPropIndex := nCurrentPropIndex + 1;
	aSpecPoints[i].X := DINT_TO_REAL(refCmdData.n32Data[nCurrentPropIndex]);
	nCurrentPropIndex := nCurrentPropIndex + 1;
	aSpecPoints[i].Y := DINT_TO_REAL(refCmdData.n32Data[nCurrentPropIndex]);
	nCurrentPropIndex := nCurrentPropIndex + 1;
	aSpecPoints[i].Z := DINT_TO_REAL(refCmdData.n32Data[nCurrentPropIndex]);
END_FOR

//WasteChannels
nCurrentPropIndex := nCurrentPropIndex + 1;
IF refCmdData.n32Data[nCurrentPropIndex] >= 1 AND refCmdData.n32Data[nCurrentPropIndex] <= cMaxWasteChannels THEN
	nNoOfWasteChannels := DINT_TO_USINT(refCmdData.n32Data[nCurrentPropIndex]);
ELSE
	{warning 'Implement ErrorId"}
	M_SetAllProps := E_ErrorIdObjMgmt.ERRORID_InvalidNoOfSlots;
	RETURN;	
END_IF

//WasteChannels parametrieren
FOR i:= 1 TO nNoOfWasteChannels BY 1 DO
	nCurrentPropIndex := nCurrentPropIndex + 1;
	aWasteChannels[i].nNr := DINT_TO_USINT(refCmdData.n32Data[nCurrentPropIndex]);
	nCurrentPropIndex := nCurrentPropIndex + 1; 
	aWasteChannels[i].nSpecPointNr := DINT_TO_USINT(refCmdData.n32Data[nCurrentPropIndex]);
	nCurrentPropIndex := nCurrentPropIndex + 1;
	aWasteChannels[i].nPumpNr := DINT_TO_USINT(refCmdData.n32Data[nCurrentPropIndex]);
	nCurrentPropIndex := nCurrentPropIndex + 1;
	aWasteChannels[i].nBottleNr := DINT_TO_USINT(refCmdData.n32Data[nCurrentPropIndex]);
END_FOR

//LiquidChannels
nCurrentPropIndex := nCurrentPropIndex + 1;
IF refCmdData.n32Data[nCurrentPropIndex] >= 1 AND refCmdData.n32Data[nCurrentPropIndex] <= cMaxLiquidChannels THEN
	nNoOfLiquidChannels := DINT_TO_USINT(refCmdData.n32Data[nCurrentPropIndex]);
ELSE
	{warning 'Implement ErrorId"}
	M_SetAllProps := E_ErrorIdObjMgmt.ERRORID_InvalidNoOfSlots;
	RETURN;	
END_IF

//LiquidChannels parametrieren
FOR i:= 1 TO nNoOfLiquidChannels BY 1 DO
	nCurrentPropIndex := nCurrentPropIndex + 1;
	aLiquidChannels[i].nNr := DINT_TO_USINT(refCmdData.n32Data[nCurrentPropIndex]);
	nCurrentPropIndex := nCurrentPropIndex + 1;
	aLiquidChannels[i].nSlotNr := DINT_TO_USINT(refCmdData.n32Data[nCurrentPropIndex]);
	nCurrentPropIndex := nCurrentPropIndex + 1;
	aLiquidChannels[i].nWasteCh := DINT_TO_USINT(refCmdData.n32Data[nCurrentPropIndex]);
	nCurrentPropIndex := nCurrentPropIndex + 1;
	aLiquidChannels[i].nBottleNr := DINT_TO_USINT(refCmdData.n32Data[nCurrentPropIndex]);
END_FOR

nNoOfProps := nCurrentPropIndex + 1;
END_METHOD

METHOD M_SetSingleProp : ERRORID
VAR_INPUT
	refCmdData : REFERENCE TO  ST_CmdData;
END_VAR
VAR
	i : UINT;
	nIndex					: UINT;
	nIndexSlots 		 	: UINT;
	nIndexSpecPoints 	 	: UINT;
	nIndexWasteChannels  	: UINT;
	nIndexLiquidChannels 	: UINT;
	nValue					: USINT;
END_VAR
nIndexSlots := nSpecPropIndex;
nIndexSpecPoints := nIndexSlots + nNoOfSlots * 5 + 1;
nIndexWasteChannels := nIndexSpecPoints + nNoOfSpecPoints * 3 + 1;
nIndexLiquidChannels := nIndexWasteChannels + nNoOfWasteChannels * 4 + 1;

//Section: Slots
IF refCmdData.aHeader[1] > nIndexSlots AND refCmdData.aHeader[1] < nIndexSpecPoints THEN
	FOR i:= 1 TO nNoOfSlots BY 1 DO
		//ersten Index innerhalb der Section ermitteln
		nIndex := nIndexSlots + ((i - 1) * 5) + 1;
		IF refCmdData.aHeader[1] = nIndex THEN
			M_SetSingleProp := E_ErrorIdCmd.ERRORID_InvalidProperty; //SlotNr darf nicht verändert werden
			RETURN;
		ELSIF refCmdData.aHeader[1] = nIndex + 1 THEN
			aSlots[i].P_rRelPosX := DINT_TO_REAL(refCmdData.n32Data[0]);
		ELSIF refCmdData.aHeader[1] = nIndex + 2 THEN
			aSlots[i].P_rRelPosY := DINT_TO_REAL(refCmdData.n32Data[0]);
		ELSIF refCmdData.aHeader[1] = nIndex + 3 THEN
			aSlots[i].P_rRelPosZ := DINT_TO_REAL(refCmdData.n32Data[0]);
		ELSIF refCmdData.aHeader[1] = nIndex + 4 THEN
			aSlots[i].P_rDepth := DINT_TO_REAL(refCmdData.n32Data[0]);
		END_IF
	END_FOR
//Section: SpePoints
ELSIF refCmdData.aHeader[1] > nIndexSpecPoints AND refCmdData.aHeader[1] < nIndexWasteChannels THEN
	FOR i:= 1 TO nNoOfSpecPoints BY 1 DO
		//ersten Index innerhalb der Section ermitteln
		nIndex := nIndexSpecPoints + ((i - 1) * 3) + 1;
		IF refCmdData.aHeader[1] = nIndex THEN
			aSpecPoints[i].X := DINT_TO_REAL(refCmdData.n32Data[0]);
		ELSIF refCmdData.aHeader[1] = nIndex + 1 THEN
			aSpecPoints[i].Y := DINT_TO_REAL(refCmdData.n32Data[0]);
		ELSIF refCmdData.aHeader[1] = nIndex + 2 THEN
			aSpecPoints[i].Z := DINT_TO_REAL(refCmdData.n32Data[0]);
		END_IF
	END_FOR
//Section WasteChannels
ELSIF refCmdData.aHeader[1] > nIndexWasteChannels AND refCmdData.aHeader[1] < nIndexLiquidChannels THEN
	FOR i:= 1 TO nNoOfWasteChannels BY 1 DO
		//ersten Index innerhalb der Section ermitteln
		nIndex := nIndexWasteChannels + ((i - 1) * 4) + 1;
		IF refCmdData.aHeader[1] = nIndex THEN
			M_SetSingleProp := E_ErrorIdCmd.ERRORID_InvalidProperty; //WasteChannelNr darf nicht verändert werden
			RETURN;
		ELSIF refCmdData.aHeader[1] = nIndex + 1 THEN
			M_SetSingleProp := E_ErrorIdCmd.ERRORID_InvalidProperty; //AssignedSpecPointNr darf nicht verändert werden
			RETURN;
		ELSIF refCmdData.aHeader[1] = nIndex + 2 THEN
			nValue := DINT_TO_USINT(refCmdData.n32Data[0]);
			IF nValue > 0 AND nValue <= cNoOfPumps THEN
				aWasteChannels[i].nPumpNr := nValue;
			ELSE
				M_SetSingleProp := E_ErrorIdObjMgmt.ERRORID_InvalidPumpNumber;
				RETURN;					
			END_IF
		ELSIF refCmdData.aHeader[1] = nIndex + 3 THEN
			nValue := DINT_TO_USINT(refCmdData.n32Data[0]);
			IF nValue > 0 AND nValue <= cNoOfWasteBottles THEN
				aWasteChannels[i].nBottleNr := nValue;
			ELSE
				M_SetSingleProp := E_ErrorIdObjMgmt.ERRORID_InvalidWastebottle;
				RETURN;					
			END_IF
		END_IF
	END_FOR
//Section LiquidChannels
ELSIF refCmdData.aHeader[1] > nIndexLiquidChannels AND refCmdData.aHeader[1] < nNoOfProps THEN
	FOR i:= 1 TO nNoOfLiquidChannels BY 1 DO
		//ersten Index innerhalb der Section ermitteln
		nIndex := nIndexLiquidChannels + ((i - 1) * 4) + 1;
		IF refCmdData.aHeader[1] = nIndex THEN
			M_SetSingleProp := E_ErrorIdCmd.ERRORID_InvalidProperty; //WasteChannelNr darf nicht verändert werden
			RETURN;
		ELSIF refCmdData.aHeader[1] = nIndex + 1 THEN
			M_SetSingleProp := E_ErrorIdCmd.ERRORID_InvalidProperty; //AssignedSpecPointNr darf nicht verändert werden
			RETURN;
		ELSIF refCmdData.aHeader[1] = nIndex + 2 THEN
			M_SetSingleProp := E_ErrorIdCmd.ERRORID_InvalidProperty; //AssignedSpecPointNr darf nicht verändert werden
			RETURN;
		ELSIF refCmdData.aHeader[1] = nIndex + 3 THEN
			nValue := DINT_TO_USINT(refCmdData.n32Data[0]);
			IF nValue > 0 AND nValue <= cNoOfLiquidBottles THEN
				aLiquidChannels[i].nBottleNr := nValue;
			ELSE
				M_SetSingleProp := E_ErrorIdObjMgmt.ERRORID_InvalidLiquidbottle;
				RETURN;					
			END_IF
		END_IF
	END_FOR
ELSE
	M_SetSingleProp := SUPER^.M_SetSingleProp(refCmdData);
END_IF
END_METHOD

METHOD M_Stop : ERRORID
VAR_INPUT
END_VAR
IF bFillLiquid AND nStateA_FillEmptyLiquid < 70 THEN
	nStateA_FillEmptyLiquid := 70;
END_IF

IF bEmptyLiquid AND nStateA_FillEmptyLiquid < 70 THEN
	nStateA_FillEmptyLiquid := 70;
END_IF
END_METHOD

END_FUNCTION_BLOCK

// ---- Objects/Targets/Active/FB_CustomUnitType2.TcPOU
FUNCTION_BLOCK FB_CustomUnitType2 EXTENDS FB_ActiveTarget
VAR
	bLevelSensor		AT %I* : BOOL;
	
	//Spec-Properties
	nPumpNrWaste		: USINT;
	nBottleNrWaste 		: USINT;
	
	//****************************************Aktionvariablen****************************************************
	
	//Action: "SuckOff"
	bSuckOff			: BOOL;
	nStateA_SuckOff		: USINT;
	bSuckOff_On			: BOOL;
	tSuckOffTime		: TIME;
	tmrSuckOffTime		: TON;
	
	//Empty (keine von außen ausführbare Action)
	bEmpty				: BOOL;
	nStateA_Empty		: USINT;
	tmrEmptyTimout		: TON;
	
END_VAR

IF bInitFB THEN
	bInitFB := FALSE;
	//Fehlerstruktur vorausfüllen
	stError.ObjectId := nObjectID;
	stError.HardwareGrp := E_HardwareGrp.Nothing;
	stError.POU := E_POU.POU_FB_CustomUnitType2;
END_IF

CASE eCurrentState OF
	E_MachineState.MACHINESTATE_Idle:

	IF MainDispacher.eCurrentMode = E_MachineMode.MACHINEMODE_Manu OR MainDispacher.eCurrentMode = E_MachineMode.MACHINEMODE_Auto THEN
		IF MainDispacher.eCurrentState <> E_MachineState.MACHINESTATE_Error THEN
			IF bIsInit THEN
				IF NOT bLevelSensor THEN 	//Leeren
					bEmpty := TRUE;
					bBusy := TRUE;
					eCurrentState := E_MachineState.MACHINESTATE_Active;	
				END_IF
			END_IF
		END_IF
	END_IF
	
	E_MachineState.MACHINESTATE_Active:
	
	IF bEmpty THEN //Ist nur eine interne Action, welche niemals in Error geht?
		A_Empty();
		IF nStateA_Empty >= 80 THEN
			IF nStateA_Empty >= 99 THEN
				bError := TRUE;
			END_IF
			bEmpty := FALSE;
			nStateA_Empty := 0;
		END_IF
	END_IF
	
	IF bSuckOff THEN
		A_SuckOff();
		IF nStateA_SuckOff >= 80 THEN
			IF nStateA_SuckOff >= 99 THEN
				bError := TRUE;	
			END_IF
			bSuckOff := FALSE;
			nStateA_SuckOff := 0;
		END_IF
	END_IF
	
	IF NOT (bSuckOff OR bEmpty) THEN
		bBusy := FALSE;
		eCurrentState := E_MachineState.MACHINESTATE_Idle;
	END_IF
	
	E_MachineState.MACHINESTATE_Reset:
		bError := FALSE;
		
END_CASE

IF bError THEN
	eCurrentState := E_MachineState.MACHINESTATE_Error;
	bBusy := FALSE;
	aPumps[nPumpNrWaste].M_Off();
END_IF

//Prozessdaten aktualisieren
stProcessData.nObjId := nObjectID;
stProcessData.n32Data[0] := BOOL_TO_DINT(bIsInit);
stProcessData.n32Data[1] := eCurrentState;
stProcessData.n32Data[2] := stError.ErrorId;
aObjProcData[nNotifyId] := stProcessData;

ACTION A_Empty:
IF nStateA_Empty = 0 THEN
	stError.ErrorId := M_CheckBottles();
	IF stError.ErrorId > 0 THEN
		stError.POUState := nStateA_Empty;
		nStateA_Empty := 99;
	ELSE
		aPumps[nPumpNrWaste].M_On();
		tmrEmptyTimout(IN:= TRUE, PT:= T#15S);
		nStateA_Empty := 1;		
	END_IF
ELSIF nStateA_Empty = 1 THEN //Warten auf Timer und Wastepumpe ausschalten
	tmrEmptyTimout();
	IF tmrEmptyTimout.Q THEN
		tmrEmptyTimout(IN:= FALSE);
		aPumps[nPumpNrWaste].M_Off();
		IF NOT bLevelSensor THEN
			aPumps[nPumpNrWaste].M_Off();
			stError.ErrorId := ERRORID_TimeOutSuckOffLiquid;
			stError.POUState := nStateA_Empty;
			nStateA_Empty := 99;
		ELSE
			nStateA_Empty := 80;
		END_IF
	END_IF
ELSIF nStateA_Empty = 70 THEN
	tmrEmptyTimout(IN:= FALSE);
	nStateA_Empty := 80;
END_IF

//Errorhandling
IF nStateA_Empty = 99 THEN
	stError.Cmd := E_Action.ACTION_EmptyWaste;
	stError.POUAction := E_POUACT.POUACT_A_EmptyWaste;
	fbErrorList.M_Add(stError);
END_IF
END_ACTION

ACTION A_SuckOff:
CASE nStateA_SuckOff OF
	0:	//Ventil und Pumpe einschalten
		IF bSuckOff_On THEN
			aPumps[nPumpNrWaste].M_On();
			IF tSuckOffTime > T#0S THEN
				nStateA_SuckOff := 1;
			ELSE
				nStateA_SuckOff := 80;
			END_IF
		ELSE
			nStateA_SuckOff := 2;
		END_IF
		tmrSuckOffTime(IN:= FALSE);
	
	1:	//Time
		tmrSuckOffTime(IN:= TRUE, PT:= tSuckOffTime);
		IF tmrSuckOffTime.Q THEN
			nStateA_SuckOff := 2;
		END_IF
	
	2:	//Ausschalten
		aPumps[nPumpNrWaste].M_Off();
		nStateA_SuckOff := 80;
		
	70:	//Abbrechen
		aPumps[nPumpNrWaste].M_Off();
		nStateA_SuckOff := 80;
		
END_CASE
END_ACTION

METHOD FB_init : BOOL
VAR_INPUT
	bInitRetains : BOOL; // if TRUE, the retain variables are initialized (warm start / cold start)
	bInCopyCode : BOOL;  // if TRUE, the instance afterwards gets moved into the copy code (online change)
END_VAR
eObjectType := E_ObjectType.OBJECTTYPE_CustomUnitType2;
eObjectGroup := E_ObjectGroup.OBJECTGROUP_Target OR E_ObjectGroup.OBJECTGROUP_Device;
END_METHOD

METHOD M_CancelAction
VAR_INPUT
	eAction : E_Action;
END_VAR
IF eAction = E_Action.ACTION_SuckOff THEN
	IF bSuckOff AND nStateA_SuckOff < 70 THEN
		nStateA_SuckOff := 70;
	END_IF
END_IF
END_METHOD

METHOD M_CheckAction : ERRORID
VAR_INPUT
	refActionData 	: REFERENCE TO ST_ActionData;
	pCorrelObject	: POINTER TO FB_Object;
END_VAR
IF refActionData.eAction = E_Action.ACTION_SuckOff THEN
	//BottleState prüfen
	M_CheckAction := M_CheckBottles();
ELSE
	M_CheckAction := SUPER^.M_CheckAction(refActionData,pCorrelObject);
END_IF
END_METHOD

METHOD M_CheckBottles : ERRORID
VAR_INPUT
END_VAR
//Wastebottle OK?
IF nBottleNrWaste > 0 THEN
	IF NOT aSensWasteBottle[nBottleNrWaste] THEN //Voll
		M_CheckBottles := E_ErrorIdCmd.ERRORID_WasteBottleFull;
		RETURN;
	END_IF
END_IF
END_METHOD

METHOD M_CheckProcDataType : BOOL
VAR_INPUT
	eProcDataType : E_ProcDataType;
END_VAR
END_METHOD

METHOD M_ExeAction : ERRORID
VAR_INPUT
	refActionData : REFERENCE TO ST_ActionData;	
END_VAR
IF refActionData.eAction = E_Action.ACTION_Init THEN
	bIsInit := TRUE;
	RETURN;
ELSIF refActionData.eAction = E_Action.ACTION_SuckOff THEN
	
	IF NOT aSensWasteBottle[nBottleNrWaste] THEN
		M_ExeAction := E_ErrorIdCmd.ERRORID_WasteBottleFull;
		RETURN;
	END_IF
	
	nStateA_SuckOff := 0;
	bSuckOff_On := DINT_TO_BOOL(refActionData.aParams[2]);
	tSuckOffTime := DINT_TO_TIME(refActionData.aParams[3]);
	bSuckOff := TRUE;
	
ELSE
	M_ExeAction := E_ErrorIdCmd.ERRORID_InvalidAction;
	RETURN;
END_IF
bBusy := TRUE;
eCurrentState:= E_MachineState.MACHINESTATE_Active;
END_METHOD

METHOD M_GetActionBusy : BOOL
VAR_INPUT
	eAction : E_Action;
END_VAR
IF eAction = E_Action.ACTION_SuckOff THEN
	M_GetActionBusy := bSuckOff;
END_IF
END_METHOD

METHOD M_GetAllProps : ERRORID
VAR_INPUT
	refCmdData : REFERENCE TO  ST_CmdData;
END_VAR
SUPER^.M_GetAllProps(refCmdData); 
nCurrentPropIndex := nCurrentPropIndex + 1;
refCmdData.n32Data[nCurrentPropIndex] := nPumpNrWaste;
nCurrentPropIndex := nCurrentPropIndex + 1;
refCmdData.n32Data[nCurrentPropIndex] := nBottleNrWaste;
END_METHOD

METHOD M_GetProcData : DINT
VAR_INPUT
	eProcDataType : E_ProcDataType;
END_VAR
END_METHOD

METHOD M_Reset
bError := FALSE;
bBusy := FALSE;
eCurrentState := E_MachineState.MACHINESTATE_Idle;
END_METHOD

METHOD M_SetAllProps : ERRORID
VAR_INPUT
	refCmdData : REFERENCE TO  ST_CmdData;
END_VAR

VAR
	i : UINT;
END_VAR
M_SetAllProps := SUPER^.M_SetAllProps(refCmdData);

IF M_SetAllProps > 0 THEN
	RETURN;
END_IF

nCurrentPropIndex := nCurrentPropIndex + 1;
nSpecPropIndex := nCurrentPropIndex;

nPumpNrWaste := DINT_TO_USINT(refCmdData.n32Data[nCurrentPropIndex]);
IF NOT (nPumpNrWaste > 0 AND nPumpNrWaste <= cNoOfPumps) THEN
	M_SetAllProps := E_ErrorIdObjMgmt.ERRORID_InvalidPumpNumber;
	RETURN;
END_IF

nCurrentPropIndex := nCurrentPropIndex + 1;
nBottleNrWaste := DINT_TO_USINT(refCmdData.n32Data[nCurrentPropIndex]);
IF NOT (nBottleNrWaste > 0 AND nBottleNrWaste <= cNoOfWasteBottles) THEN
	M_SetAllProps := E_ErrorIdObjMgmt.ERRORID_InvalidWastebottle;
	RETURN;
END_IF

nNoOfProps := nCurrentPropIndex + 1;
END_METHOD

METHOD M_SetSingleProp : ERRORID
VAR_INPUT
	refCmdData : REFERENCE TO  ST_CmdData;
END_VAR

VAR
	value : USINT;
END_VAR
IF nSpecPropIndex = refCmdData.aHeader[1] THEN
	//PumpNrWaste
	IF refCmdData.n32Data[0] > 0 AND refCmdData.n32Data[0] <= cNoOfPumps THEN
		nPumpNrWaste := DINT_TO_USINT(refCmdData.n32Data[0]);
	ELSE
		M_SetSingleProp := E_ErrorIdObjMgmt.ERRORID_InvalidPumpNumber;
	END_IF
ELSIF nSpecPropIndex + 1 = refCmdData.aHeader[1] THEN
	//BottleNrWaste
	IF refCmdData.n32Data[0] > 0 AND refCmdData.n32Data[0] <= cNoOfWasteBottles THEN
		nBottleNrWaste := DINT_TO_USINT(refCmdData.n32Data[0]);
	ELSE
		M_SetSingleProp := E_ErrorIdObjMgmt.ERRORID_InvalidWastebottle;
	END_IF	
ELSE
	M_SetSingleProp := SUPER^.M_SetSingleProp(refCmdData);
END_IF
END_METHOD

METHOD M_Stop : ERRORID
VAR_INPUT
END_VAR
IF bSuckOff AND nStateA_SuckOff < 70 THEN
	nStateA_SuckOff:= 70;
END_IF
END_METHOD

END_FUNCTION_BLOCK

// ---- Objects/Targets/Active/FB_TrayTransporter.TcPOU
FUNCTION_BLOCK FB_TrayTransporter EXTENDS FB_ActiveTarget IMPLEMENTS I_SlotTarget

VAR
	fbSlotList			: FB_SlotList;
	pSlot				: POINTER TO FB_Slot;
	nNumberOfSlots		: UINT;
	nFirstSlotPropIndex	: UINT;	//erster Index für Slots (benötigt in M_SetSingleProps)
	nLastSlotPropIndex	: UINT;	//letzte Index für Slots (benötigt in M_SetSingleProps)
	
	pTraySlot			: POINTER TO FB_Slot;
	
	nTemp				: DINT;

	//Hardware-Verküpfung
	pSliderRef			: POINTER TO FB_HwRefNanotecPD;
	pDrivingPinRefLeft	: POINTER TO FB_HwRefTMCM1140;
	pDrivingPinRefRight	: POINTER TO FB_HwRefTMCM1140;
	pTrayLock			: POINTER TO FB_HwRefTrayLock;
	bReadyFlagLeft		AT %I* : BOOL;
	bReadyFlagRight		AT %I* : BOOL;
	
	//Spec-Properties
	nOffsetLeftDrivingPin	: DINT;
	nOffsetRightDrivingPin	: DINT;
	nDrivingPinThickness	: DINT;
	nTransferPosLeft		: DINT;
	nTransferPosRight		: DINT;
	nSafePosLeft			: DINT;
	nSafePosRight			: DINT;
	nTrayLength				: DINT;
	nHollowDistance			: DINT;
	nHollowWidth			: DINT;
	
	//****************************************Aktionvariablen****************************************************
	
	//Action: "Init"
	fbSliderPower 			: FB_NanotecPD_Power;
	fbDrivingPinLeftPower 	: FB_TMCM1140_Power;
	fbDrivingPinRightPower 	: FB_TMCM1140_Power;
	fbSliderHome			: FB_NanotecPD_Home;
	fbDrivingPinLeftHome	: FB_TMCM1140_Home;
	fbDrivingPinRightHome	: FB_TMCM1140_Home;
	
	//Action: "MoveTrayTransporter"
	bMoveSlider			: BOOL;
	fbMoveSlider 		: FB_NanotecPD_Move;
	nStateA_MoveSlider 	: USINT;
	
	nMoveSliderPosition	: DINT;
	nMoveSliderSpeed	: DINT;
	
	//Action: "TurnDrivingPin"
	bTurnDrivingPin			: BOOL;
	nStateA_TurnDrivingPin	: USINT;
	eTurnDrivingPinSel		: E_DrivingPinSelection;
	eTurnDrivingPinCtrl		: E_DrivingPinCtrl;
	fbTurnDrivingPinLeft	: FB_TMCM1140_Move;
	fbTurnDrivingPinRight	: FB_TMCM1140_Move;
	bReHomingLeftPin		: BOOL;
	bReHomingRightPin		: BOOL;
	
	//Action: "LockUnlock"
	bLockUnlock				: BOOL;
	nStateA_LockUnlock		: USINT;
	eLockCtrl				: E_LockCtrl;
	fbTrayLockCtrl			: FB_HwTrayLockControl;

END_VAR

IF bInitFB THEN
	bInitFB := FALSE;
	F_CreateLinkedListHnd(ADR(aNodes), SIZEOF(aNodes), hList);
	stError.ObjectId := nObjectID;
	stError.HardwareGrp := E_HardwareGrp.Nothing;
	stError.POU := E_POU.POU_FB_TrayTransporter;
END_IF

CASE eCurrentState OF
	E_MachineState.MACHINESTATE_Active:
		IF bInit THEN
			A_Init();
			IF nStateA_Init >= 80 THEN
				bIsInit := TRUE;
				IF nStateA_Init >= 99 THEN
					bError := TRUE;
					bIsInit := FALSE;
				END_IF
				bInit := FALSE;
				nStateA_Init := 0;
				M_RemoveListEntry(nSearchValue:= E_Action.ACTION_Init);
			END_IF
		END_IF
		
		IF bMoveSlider THEN
			A_MoveSlider();
			IF nStateA_MoveSlider >= 80 THEN
				IF bStop THEN
					bCanceled := TRUE;
				END_IF
				IF nStateA_MoveSlider >= 99 THEN
					bError := TRUE;
				END_IF
				bMoveSlider := FALSE;
				nStateA_MoveSlider := 0;
				M_RemoveListEntry(nSearchValue:= E_Action.ACTION_MoveTrayTransporter);
			END_IF
		END_IF
		
		IF bTurnDrivingPin THEN
			A_TurnDrivingPin();
			IF nStateA_TurnDrivingPin >= 80 THEN
				IF bStop THEN
					bCanceled := TRUE;
				END_IF
				IF nStateA_TurnDrivingPin >= 99 THEN
					bError := TRUE;
				END_IF
				bTurnDrivingPin := FALSE;
				nStateA_TurnDrivingPin := 0;
				M_RemoveListEntry(nSearchValue:= E_Action.ACTION_TurnDrivingPin);
			END_IF
		END_IF
		
		IF bLockUnlock THEN
			A_LockUnlock();
			IF nStateA_LockUnlock >= 80 THEN
				IF bStop THEN
					bCanceled := TRUE;
				END_IF
				IF nStateA_LockUnlock >= 99 THEN
					bError := TRUE;
				END_IF
				bLockUnlock := FALSE;
				nStateA_LockUnlock := 0;
				M_RemoveListEntry(nSearchValue:= E_Action.ACTION_LockUnlock);
			END_IF
		END_IF
	
		IF hList.nCount = 0 THEN
			eCurrentState := E_MachineState.MACHINESTATE_Ready;
		END_IF

		IF bError  THEN
			eCurrentState := E_MachineState.MACHINESTATE_Error;
		END_IF
		
	E_MachineState.MACHINESTATE_Reset:
			nStateA_Init := 0;
			nStateA_Reset := 0;
			bBusy := FALSE;
			bError := FALSE;
			bStop := FALSE;
			bStopAllOnError := FALSE;
			fbList.A_Reset(hList:= hList);
			nErrorId := 0;
			stError.Cmd := 0;
			stError.ErrorId := 0;
			eCurrentState := E_MachineState.MACHINESTATE_Idle;

	E_MachineState.MACHINESTATE_Ready:
		bBusy := FALSE;
		bStop := FALSE;
		eCurrentState := E_MachineState.MACHINESTATE_Idle;
	
	E_MachineState.MACHINESTATE_Error:
		bBusy := FALSE;	
		bStop := FALSE;
END_CASE

//Prozessdaten aktualisieren
stProcessData.nObjId := nObjectID;
bIsInit := TRUE;

stProcessData.n32Data[1] := eCurrentState;
stProcessData.n32Data[2] := stError.ErrorId;
stProcessData.n32Data[3] := pSliderRef^.P_nCurrentRealPos;
IF pDrivingPinRefLeft > 0 THEN
	bIsInit := bIsInit AND pDrivingPinRefLeft^.P_bIsHomed;
	nTemp := pDrivingPinRefLeft^.P_nCurrentPosReal;
	IF nTemp >= -10 AND nTemp <= 10 THEN //horizontal
		stProcessData.n32Data[4] := E_DrivingPinState.Horizontal;	
	ELSIF nTemp >= 890 AND nTemp <= 910 THEN //vertikal
		stProcessData.n32Data[4] := E_DrivingPinState.Vertical;
	ELSE
		stProcessData.n32Data[4] := E_DrivingPinState.UNDEFINED;
	END_IF
END_IF

IF pDrivingPinRefRight > 0 THEN
	bIsInit := bIsInit AND pDrivingPinRefRight^.P_bIsHomed;
	IF nTemp >= -10 AND nTemp <= 10 THEN //horizontal
		stProcessData.n32Data[5] := E_DrivingPinState.Horizontal;	
	ELSIF nTemp >= 890 AND nTemp <= 910 THEN //vertikal
		stProcessData.n32Data[5] := E_DrivingPinState.Vertical;
	ELSE
		stProcessData.n32Data[5] := E_DrivingPinState.UNDEFINED;
	END_IF
END_IF

bIsInit := bIsInit AND pSliderRef^.P_bIsHomed;
stProcessData.n32Data[0] := BOOL_TO_DINT(bIsInit);

IF pTrayLock^.eCurrentState = E_LockState.Locked THEN
	stProcessData.n32Data[6] := E_LockCtrl.Lock;
ELSIF pTrayLock^.eCurrentState = E_LockState.Unlocked THEN
	stProcessData.n32Data[6] := E_LockCtrl.Unlock;
ELSE
	stProcessData.n32Data[6] := 99;
END_IF

aObjProcData[nNotifyId] := stProcessData;

ACTION A_Init:
IF nStateA_Init = 0 THEN	//Power
	{IF defined (TrayTransporterL)}
	pDrivingPinRefLeft^.P_bIsHomed := FALSE;
	fbDrivingPinLeftPower(pHwRef:= pDrivingPinRefLeft, bExecute:= TRUE);
	fbSliderPower(pHwRef := pSliderRef, bExecute := TRUE);
	IF NOT (fbDrivingPinLeftPower.bBusy OR fbSliderPower.bBusy) THEN
		IF fbDrivingPinLeftPower.bError THEN
			stError.ErrorId := fbDrivingPinLeftPower.nErrorId;
			stError.POUState := nStateA_Init;
			//stError.HardwareGrp := pDrivingPinRefLeft^.P_stHardwareId.eGroup;
			//stError.HardwareNr := pDrivingPinRefLeft^.P_stHardwareId.nItem;
			nStateA_Init := 99;
		ELSIF fbSliderPower.bError THEN
			stError.ErrorId := fbSliderPower.nErrorId;
			stError.POUState := nStateA_Init;
			nStateA_Init := 99;
		ELSE
			nStateA_Init := 1;
		END_IF
		fbDrivingPinLeftPower(pHwRef:= pDrivingPinRefLeft, bExecute:= FALSE);
		fbSliderPower(pHwRef := pSliderRef, bExecute := FALSE);
	END_IF
	
	{ELSIF defined (TrayTransporterR)}
	pDrivingPinRefRight^.P_bIsHomed := FALSE;
	fbDrivingPinRightPower(pHwRef:= pDrivingPinRefRight, bExecute:= TRUE);
	fbSliderPower(pHwRef := pSliderRef, bExecute := TRUE);
	IF NOT (fbDrivingPinRightPower.bBusy OR fbSliderPower.bBusy) THEN
		IF fbDrivingPinRightPower.bError THEN
			stError.ErrorId := fbDrivingPinRightPower.nErrorId;
			stError.POUState := nStateA_Init;
			nStateA_Init := 99;
		ELSIF fbSliderPower.bError THEN
			stError.ErrorId := fbSliderPower.nErrorId;
			stError.POUState := nStateA_Init;
			nStateA_Init := 99;
		ELSE
			nStateA_Init := 1;
		END_IF
		fbDrivingPinRightPower(pHwRef:= pDrivingPinRefRight, bExecute:= FALSE);
		fbSliderPower(pHwRef := pSliderRef, bExecute := FALSE);
	END_IF
	
	{ELSIF defined (TrayTransporterLR)}
	fbDrivingPinLeftPower(pHwRef:= pDrivingPinRefLeft ,bExecute:= TRUE);
	fbDrivingPinRightPower(pHwRef:= pDrivingPinRefRight, bExecute:= TRUE);
	fbSliderPower(pHwRef := pSliderRef, bExecute := TRUE);
	IF NOT (fbDrivingPinLeftPower.bBusy OR fbDrivingPinRightPower.bBusy OR fbSliderPower.bBusy) THEN
		IF fbDrivingPinLeftPower.bError THEN
			stError.ErrorId := fbDrivingPinLeftPower.nErrorId;
			stError.POUState := nStateA_Init;
			nStateA_Init := 99;
		ELSIF fbDrivingPinRightPower.bError THEN
			stError.ErrorId := fbDrivingPinRightPower.nErrorId;
			stError.POUState := nStateA_Init;
			nStateA_Init := 99;
		ELSIF fbSliderPower.bError THEN
			stError.ErrorId := fbSliderPower.nErrorId;
			stError.POUState := nStateA_Init;
			nStateA_Init := 99;
		ELSE
			nStateA_Init := 1;
		END_IF
		fbDrivingPinLeftPower(pHwRef:= pDrivingPinRefLeft, bExecute:= FALSE);
		fbDrivingPinRightPower(pHwRef:= pDrivingPinRefRight, bExecute:= FALSE);
		fbSliderPower(pHwRef:= pSliderRef, bExecute := FALSE);
	END_IF
	{END_IF}
	pSliderRef^.P_bIsHomed := FALSE;
	
ELSIF nStateA_Init = 1 THEN //Homing Driving pins
	{IF defined (TrayTransporterL)}
	fbDrivingPinLeftHome(pHwRef:= pDrivingPinRefLeft, bExecute:= TRUE, bStop:= bStop);
	IF NOT fbDrivingPinLeftHome.bBusy THEN
		IF fbDrivingPinLeftHome.bError THEN
			stError.ErrorId := fbDrivingPinLeftHome.nErrorId;
			stError.POUState := nStateA_Init;
			nStateA_Init := 99;
		ELSE
			nStateA_Init := 2;
		END_IF
		fbDrivingPinLeftHome(pHwRef:= pDrivingPinRefLeft, bExecute:= FALSE);
	END_IF
	{ELSIF defined (TrayTransporterR)}
	fbDrivingPinRightHome(pHwRef:= pDrivingPinRefRight, bExecute:= TRUE, bStop:= bStop);
	IF NOT fbDrivingPinRightHome.bBusy THEN
		IF fbDrivingPinRightHome.bError THEN
			stError.ErrorId := fbDrivingPinRightHome.nErrorId;
			stError.POUState := nStateA_Init;
			nStateA_Init := 99;
		ELSE
			nStateA_Init := 2;
		END_IF
		fbDrivingPinRightHome(pHwRef:= pDrivingPinRefRight, bExecute:= FALSE);
	END_IF
	
	{ELSIF defined (TrayTransporterLR)}
	fbDrivingPinLeftHome(pHwRef:= pDrivingPinRefLeft, bExecute:= TRUE, bStop:= bStop);
	fbDrivingPinRightHome(pHwRef:= pDrivingPinRefRight, bExecute:= TRUE,  bStop:= bStop);
	IF NOT (fbDrivingPinLeftHome.bBusy OR fbDrivingPinRightHome.bBusy) THEN
		IF fbDrivingPinLeftHome.bError THEN
			stError.ErrorId := fbDrivingPinLeftHome.nErrorId;
			stError.POUState := nStateA_Init;
			nStateA_Init := 99;
		ELSIF fbDrivingPinRightHome.bError THEN
			stError.ErrorId := fbDrivingPinRightHome.nErrorId;
			stError.POUState := nStateA_Init;
			nStateA_Init := 99;
		ELSE
			nStateA_Init := 2;
		END_IF
		fbDrivingPinLeftHome(pHwRef:= pDrivingPinRefLeft, bExecute:= FALSE);
		fbDrivingPinRightHome(pHwRef:= pDrivingPinRefRight, bExecute:= FALSE);
	END_IF
	{END_IF}
	
ELSIF nStateA_Init = 2 THEN //Homing slider
	fbSliderHome(pHwRef := pSliderRef, bExecute := TRUE, bStop:= bStop);
	IF NOT fbSliderHome.bBusy THEN
		IF fbSliderHome.bError THEN
			stError.ErrorId := fbSliderHome.nErrorId;
			nStateA_Init := 99;
		ELSE
			nStateA_Init := 80;
		END_IF
		fbSliderHome(pHwRef := pSliderRef, bExecute := FALSE);
	END_IF
END_IF

//Errorhandling
IF nStateA_Init = 99 THEN
	stError.Cmd := E_Action.ACTION_Init;
	stError.POUAction := E_POUACT.POUACT_A_Init;
	fbErrorList.M_Add(stError);
END_IF
END_ACTION

ACTION A_LockUnlock:
IF nStateA_LockUnlock = 0 THEN
	fbTrayLockCtrl(pHwRef:= pTrayLock, eCtrl:= eLockCtrl, bExecute:= TRUE);
	IF NOT fbTrayLockCtrl.bBusy THEN
		IF fbTrayLockCtrl.bError THEN
			stError.ErrorId := fbTrayLockCtrl.nErrorId;
			nStateA_LockUnlock := 99;
		ELSE
			nStateA_LockUnlock := 80;
		END_IF
		fbTrayLockCtrl(pHwRef:= pTrayLock, bExecute:= FALSE);
	END_IF
END_IF

//Errorhandling
IF nStateA_LockUnlock = 99 THEN
	stError.Cmd := E_Action.ACTION_LockUnlock;
	stError.POUAction := E_POUACT.POUACT_A_LockUnlock;
	fbErrorList.M_Add(stError);
END_IF
END_ACTION

ACTION A_MoveSlider:
IF nStateA_MoveSlider = 0 THEN
	fbMoveSlider(pHWRef:= pSliderRef, bStop:= bStop, bExecute := TRUE);
	IF NOT fbMoveSlider.bBusy THEN
		IF fbMoveSlider.bError THEN
			stError.ErrorId := fbMoveSlider.nErrorId;
			nStateA_MoveSlider := 99;
		ELSE
			nStateA_MoveSlider := 80;
		END_IF
		fbMoveSlider(pHWRef:= pSliderRef, bExecute := FALSE);
	END_IF
END_IF

//Errorhandling
IF nStateA_MoveSlider = 99 THEN
	stError.Cmd := E_Action.ACTION_MoveTrayTransporter;
	stError.POUAction := E_POUACT.POUACT_A_MoveSlider;
	fbErrorList.M_Add(stError);
END_IF
END_ACTION

ACTION A_TurnDrivingPin:
IF nStateA_TurnDrivingPin = 0 THEN
	CASE eTurnDrivingPinSel OF
		E_DrivingPinSelection.Left:
			fbTurnDrivingPinLeft(pHwRef:= pDrivingPinRefLeft, nSpeed:= -1, bRelative:= FALSE, bExecute:= TRUE, bStop:= bStop); 
		E_DrivingPinSelection.Right:
			fbTurnDrivingPinRight(pHwRef:= pDrivingPinRefRight, nSpeed:= -1, bRelative:= FALSE, bExecute:= TRUE, bStop:= bStop);
		E_DrivingPinSelection.Both:
			IF pDrivingPinRefLeft > 0 THEN
				fbTurnDrivingPinLeft(pHwRef:= pDrivingPinRefLeft, nSpeed:= -1, bRelative:= FALSE, bExecute:= TRUE, bStop:= bStop);
			END_IF
			IF pDrivingPinRefRight > 0 THEN
				fbTurnDrivingPinRight(pHwRef:= pDrivingPinRefRight, nSpeed:= -1, bRelative:= FALSE, bExecute:= TRUE, bStop:= bStop);	
			END_IF
	END_CASE
	
	IF NOT (fbTurnDrivingPinLeft.bBusy OR fbTurnDrivingPinRight.bBusy) THEN
		IF fbTurnDrivingPinLeft.bError THEN
			stError.ErrorId := fbTurnDrivingPinLeft.nErrorId;
			nStateA_TurnDrivingPin := 99;
		ELSIF fbTurnDrivingPinRight.bError THEN
			stError.ErrorId := fbTurnDrivingPinRight.nErrorId;
			nStateA_TurnDrivingPin := 99;
		ELSE
			nStateA_TurnDrivingPin := 80;
			IF NOT bStop THEN
				CASE eTurnDrivingPinSel OF
					E_DrivingPinSelection.Left:
						IF eTurnDrivingPinCtrl = E_DrivingPinCtrl.Horizontal THEN //HomeSwitch muss betätigt sein
							IF NOT pDrivingPinRefLeft^.P_bHomeSwitch THEN //Error
								nStateA_TurnDrivingPin := 1;
								bReHomingLeftPin := TRUE;
							END_IF
						ELSE //LimitSwitchRight muss betätigt sein
							IF NOT pDrivingPinRefLeft^.P_bRightLimitSwitch THEN //Error
								nStateA_TurnDrivingPin := 1;
								bReHomingLeftPin := TRUE;
							END_IF
						END_IF
					E_DrivingPinSelection.Right:
						IF eTurnDrivingPinCtrl = E_DrivingPinCtrl.Horizontal THEN //HomeSwitch muss betätigt sein
							IF NOT pDrivingPinRefRight^.P_bHomeSwitch THEN //Error
								nStateA_TurnDrivingPin := 1;
								bReHomingRightPin := TRUE;
							END_IF
						ELSE //LimitSwitchRight muss betätigt sein
							IF NOT pDrivingPinRefRight^.P_bRightLimitSwitch THEN //Error
								nStateA_TurnDrivingPin := 1;
								bReHomingRightPin := TRUE;
							END_IF
						END_IF
					E_DrivingPinSelection.Both:
						IF eTurnDrivingPinCtrl = E_DrivingPinCtrl.Horizontal THEN //HomeSwitches müssen betätigt sein
							IF pDrivingPinRefLeft > 0 AND_THEN NOT pDrivingPinRefLeft^.P_bHomeSwitch THEN //Error
								nStateA_TurnDrivingPin := 1;
								bReHomingLeftPin := TRUE;
							END_IF
							IF pDrivingPinRefRight > 0 AND_THEN NOT pDrivingPinRefRight^.P_bHomeSwitch THEN //Error
								nStateA_TurnDrivingPin := 1;
								bReHomingRightPin := TRUE;
							END_IF
						ELSE
							IF pDrivingPinRefLeft > 0 AND_THEN NOT pDrivingPinRefLeft^.P_bRightLimitSwitch THEN //Error
								nStateA_TurnDrivingPin := 1;
								bReHomingLeftPin := TRUE;
							END_IF
							IF pDrivingPinRefRight > 0 AND_THEN NOT pDrivingPinRefRight^.P_bRightLimitSwitch THEN //Error
								nStateA_TurnDrivingPin := 1;
								bReHomingRightPin := TRUE;
							END_IF
						END_IF
				END_CASE
			END_IF
		END_IF
		fbTurnDrivingPinLeft(pHwRef:= pDrivingPinRefLeft, bExecute:= FALSE);
		fbTurnDrivingPinRight(pHwRef:= pDrivingPinRefRight, bExecute:= FALSE);
	END_IF
ELSIF nStateA_TurnDrivingPin = 1 THEN //ReHoming pins -> danach in Error
	IF bReHomingLeftPin THEN
		fbDrivingPinLeftHome(pHwRef:= pDrivingPinRefLeft, bExecute:= TRUE);	
	END_IF
	
	IF bReHomingRightPin THEN
		fbDrivingPinRightHome(pHwRef:= pDrivingPinRefRight, bExecute:= TRUE);	
	END_IF
	
	IF NOT (fbDrivingPinLeftHome.bBusy OR fbDrivingPinRightHome.bBusy) THEN
		fbDrivingPinLeftHome(pHwRef:= pDrivingPinRefLeft, bExecute:= FALSE);
		fbDrivingPinRightHome(pHwRef:= pDrivingPinRefRight, bExecute:= FALSE);
		bReHomingLeftPin := FALSE;
		bReHomingRightPin := FALSE;
		stError.ErrorId := E_ErrorIdCmd.ERRORID_DrivingPinBlocked;
		nStateA_TurnDrivingPin := 99;
	END_IF
END_IF

//Errorhandling
IF nStateA_TurnDrivingPin = 99 THEN
	stError.Cmd := E_Action.ACTION_TurnDrivingPin;
	stError.POUAction := E_POUACT.POUACT_A_TurnDrivingPin;
	fbErrorList.M_Add(stError);
END_IF
END_ACTION

METHOD FB_init : BOOL
VAR_INPUT
	bInitRetains : BOOL; // if TRUE, the retain variables are initialized (warm start / cold start)
	bInCopyCode : BOOL;  // if TRUE, the instance afterwards gets moved into the copy code (online change)
END_VAR
eObjectType := E_ObjectType.OBJECTTYPE_TrayTransporter;
eObjectGroup := E_ObjectGroup.OBJECTGROUP_Target OR E_ObjectGroup.OBJECTGROUP_Device;
END_METHOD

METHOD M_AddChild : ERRORID
VAR_INPUT
	pObject : POINTER TO FB_Object;
	nSlotNr	: UINT;
	nIndex 	: INT;	
END_VAR

VAR
	pSlot : POINTER TO FB_Slot;
END_VAR
//In den abgeleiteten Tool-FBs wird überprüft, ob das entsprechende Objekt als Child tauglich ist
IF pObject > 0 THEN
	IF nSlotNr > 0 THEN
		pSlot := fbSlotList.M_GetAtNr(nSlotNr);
		IF pSlot > 0 THEN
			IF pSlot^.P_pChild = 0 THEN
				//Object darf selber noch an keinem Parent hängen
				IF pObject^.P_pParentObject = 0 THEN
					pSlot^.P_pChild := pObject;
					pObject^.P_pObjCollectNode := pObjCollectNode^.nodes.M_AddNewNode(pObject,nIndex);
					pObject^.M_UpdateParent();
				ELSE
					M_AddChild := E_ErrorIdObjMgmt.ERRORID_ObjectAlreadyOnAnotherParent;
				END_IF
			ELSE //Slot bereits belegt
				M_AddChild := E_ErrorIdObjMgmt.ERRORID_SlotIsAlreadyOccupied;
			END_IF		
		ELSE
			M_AddChild := E_ErrorIdObjMgmt.ERRORID_InvalidSlotNumber;			
		END_IF	
	ELSE
		M_AddChild := SUPER^.M_AddChild(pObject,nSlotNr,nIndex);
	END_IF
ELSE
	M_AddChild := E_ErrorIdObjMgmt.ERRORID_InvalidParentObject;
END_IF
END_METHOD

METHOD M_CancelAction
VAR_INPUT
	eAction : E_Action;
END_VAR
//Eine einzelne Action abzubrechen ist hier nicht implementiert.
bStop := TRUE;
END_METHOD

METHOD M_CheckAction : ERRORID
VAR_INPUT
	refActionData 	: REFERENCE TO ST_ActionData;
	pCorrelObject	: POINTER TO FB_Object;
END_VAR
IF NOT refActionData.eAction = E_Action.ACTION_MoveToTarget THEN
	M_CheckAction := E_ErrorIdCmd.ERRORID_InvalidAction;	
END_IF
END_METHOD

METHOD M_ClearAllProps
VAR_INPUT
	bIgnoreParent : BOOL; //Es wird das gesamte OD gelöscht. -> Zeiger auf Parent nicht mehr gültig!
END_VAR
fbSlotList.M_Reset();
SUPER^.M_ClearAllProps(bIgnoreParent);
END_METHOD

METHOD M_ExeAction : ERRORID
VAR_INPUT
	refActionData	: REFERENCE TO ST_ActionData;
END_VAR
IF NOT (eCurrentState = E_MachineState.MACHINESTATE_Idle OR
	eCurrentState = E_MachineState.MACHINESTATE_Active OR
	eCurrentState = E_MachineState.MACHINESTATE_Ready) THEN
	M_ExeAction := E_ErrorIdCmd.ERRORID_InvalidState;
	RETURN;
END_IF

IF bStop THEN
	M_ExeAction := E_ErrorIdCmd.ERRORID_InvalidState;
	RETURN;
END_IF

bCanceled := FALSE;

CASE refActionData.eAction OF
	E_Action.ACTION_Init:
		IF NOT bInit THEN
			bInit := TRUE;
			fbList.A_AddHeadValue(hList := hList, putValue:= E_Action.ACTION_Init);
		ELSE
			RETURN;
		END_IF
	E_Action.ACTION_MoveTrayTransporter:
		IF NOT bIsInit THEN
			M_ExeAction := E_ErrorIdCmd.ERRORID_DeviceNotInitialized;  //Error
			RETURN;
		END_IF
		
		IF bMoveSlider THEN
			M_ExeAction := E_ErrorIdCmd.ERRORID_BasicActionActive;
			RETURN;
		END_IF
		
		fbMoveSlider(pHWRef:= pSliderRef, nPosition:= refActionData.aParams[1], nSpeed:= refActionData.aParams[2], 
					bStop:= FALSE, bExecute := TRUE);
		IF fbMoveSlider.bError THEN
			M_ExeAction := fbMoveSlider.nErrorId;
			fbMoveSlider(pHWRef:= pSliderRef, bExecute := FALSE);
			RETURN;
		END_IF
		
		bMoveSlider := TRUE;
		fbList.A_AddHeadValue(hList := hList, putValue:= E_Action.ACTION_MoveTrayTransporter);
		
	E_Action.ACTION_TurnDrivingPin:
		IF NOT bIsInit THEN
			M_ExeAction := E_ErrorIdCmd.ERRORID_DeviceNotInitialized;  //Error
			RETURN;
		END_IF
		
		IF bTurnDrivingPin THEN
			M_ExeAction := E_ErrorIdCmd.ERRORID_BasicActionActive;
			RETURN;
		END_IF
		
		eTurnDrivingPinSel := DINT_TO_USINT(refActionData.aParams[1]);
		eTurnDrivingPinCtrl := DINT_TO_USINT(refActionData.aParams[2]);
		IF eTurnDrivingPinSel = E_DrivingPinSelection.Left THEN
			IF pDrivingPinRefLeft = 0 THEN
				M_ExeAction := E_ErrorIdCmd.ERRORID_DrivingPinLeftNotAvailable;
				RETURN;
			END_IF
		ELSIF eTurnDrivingPinSel = E_DrivingPinSelection.Right THEN
			IF pDrivingPinRefRight = 0 THEN
				M_ExeAction := E_ErrorIdCmd.ERRORID_DrivingPinRightNotAvailable;
				RETURN;
			END_IF
		END_IF
		
		IF eTurnDrivingPinCtrl = E_DrivingPinCtrl.Horizontal THEN
			fbTurnDrivingPinLeft.nPosition := 0;
			fbTurnDrivingPinRight.nPosition := 0;
		ELSE
			fbTurnDrivingPinLeft.nPosition := 900;
			fbTurnDrivingPinRight.nPosition := 900;
		END_IF
		
		bTurnDrivingPin := TRUE;
		fbList.A_AddHeadValue(hList := hList, putValue:= E_Action.ACTION_TurnDrivingPin);
		
	E_Action.ACTION_LockUnlock:
	
		IF bLockUnlock THEN
			M_ExeAction := E_ErrorIdCmd.ERRORID_BasicActionActive;
			RETURN;
		END_IF
		
		eLockCtrl := DINT_TO_USINT(refActionData.aParams[1]);
		bLockUnlock := TRUE;
		fbList.A_AddHeadValue(hList := hList, putValue:= E_Action.ACTION_LockUnlock);
	
	ELSE
		M_ExeAction := E_ErrorIdCmd.ERRORID_InvalidAction;	
END_CASE

bBusy := TRUE;
eCurrentState := E_MachineState.MACHINESTATE_Active;
END_METHOD

METHOD M_GetAbsPos : ST_3DPoint
VAR_INPUT
	pChildPos	: POINTER TO ST_3DPoint;
	eTargetRef 	: E_TargetRef;
	nParam1		: UINT;
 	nParam2		: UINT;
	nParam3		: USINT;
	nParam4		: USINT;
	nZLevel		: USINT;
END_VAR
VAR_OUTPUT
	nErrorId 	: ERRORID;
	lrAngle		: LREAL;
END_VAR
VAR
	stLocPos : ST_3DPoint;
	pSlot : POINTER TO FB_Slot;
END_VAR
IF eTargetRef = E_TargetRef.TARGETREF_Slot THEN
	//Slotnummer checken
	pSlot := M_GetSlot(nParam1);
	IF pSlot > 0 THEN
		stLocPos := F_Add3DPoints(pSlot^.P_stRelPos,stRelPos);
		stLocPos.Z := stLocPos.Z + stDimension.Height;
		//kann es mal sein, dass hier das ParentTarget = 0 ist?
		//ja -> bei der Workplate
		IF pChildPos > 0 THEN
			stLocPos := F_Add3DPoints(stLocPos,pChildPos^);
		END_IF
		IF pParentTarget > 0 THEN
			IF pParentSlot > 0 THEN
				M_GetAbsPos := pParentTarget^.M_GetAbsPos(pChildPos := ADR(stLocPos), eTargetRef:= E_TargetRef.TARGETREF_Slot,
															nParam1:= pParentSlot^.P_nNr,
															nParam2:= 0, nParam3:= 0,nParam4:= 0, nZLevel:= 0, lrAngle=> lrAngle,
															nErrorId=> nErrorId);		
			ELSE
				M_GetAbsPos := pParentTarget^.M_GetAbsPos(pChildPos := ADR(stLocPos), eTargetRef:= E_TargetRef.TARGETREF_LeftBottom,
																nParam1:= 0,
																nParam2:= 0, nParam3:= 0,nParam4:= 0, nZLevel:= 0,
																lrAngle => lrAngle, nErrorId=> nErrorId);
			END_IF
		ELSE
			M_GetAbsPos := stLocPos;
		END_IF		
	ELSE
		nErrorId := E_ErrorIdCmd.ERRORID_InvalidTargetSlot;
	END_IF
	
ELSE
	M_GetAbsPos := SUPER^.M_GetAbsPos(pChildPos := pChildPos, eTargetRef:= eTargetRef,
													nParam1:= nParam1,
													nParam2:= nParam2, nParam3:= nParam3, nParam4:= 0, nZLevel:= nZLevel,
													lrAngle => lrAngle, nErrorId=> nErrorId);	
END_IF
END_METHOD

METHOD M_GetActionBusy : BOOL
VAR_INPUT
	eAction : E_Action;
END_VAR
getPosPtr := 0;(* start from first node element *)
fbList.A_FindNext( hList := hList, putPosPtr := getPosPtr, putValue := eAction, getValue=>getValue, getPosPtr=>getPosPtr );
IF fbList.bOk THEN	//Eintrag wurde gefunden, d.h. Action ist noch busy
	M_GetActionBusy := TRUE;
END_IF
END_METHOD

METHOD M_GetAllProps : ERRORID
VAR_INPUT
	refCmdData : REFERENCE TO  ST_CmdData;
END_VAR

VAR
	i : UINT;
	pSlot		: POINTER TO FB_Slot;
END_VAR
SUPER^.M_GetAllProps(refCmdData);

nCurrentPropIndex := nCurrentPropIndex + 1;

refCmdData.n32Data[nCurrentPropIndex] := fbSlotList.P_nCount;

fbSlotList.M_SetCurrentToHead();

FOR i := 1 TO fbSlotList.P_nCount BY 1 DO
	pSlot := fbSlotList.M_GetNext();
	IF pSlot > 0 THEN
		nCurrentPropIndex := nCurrentPropIndex + 1;
		refCmdData.n32Data[nCurrentPropIndex] := pSlot^.P_nNr;
		nCurrentPropIndex := nCurrentPropIndex + 1;
		refCmdData.n32Data[nCurrentPropIndex] := REAL_TO_DINT(pSlot^.P_rRelPosX);
		nCurrentPropIndex := nCurrentPropIndex + 1;
		refCmdData.n32Data[nCurrentPropIndex] := REAL_TO_DINT(pSlot^.P_rRelPosY);
		nCurrentPropIndex := nCurrentPropIndex + 1;
		refCmdData.n32Data[nCurrentPropIndex] := REAL_TO_DINT(pSlot^.P_rRelPosZ);
	END_IF		
END_FOR	

nCurrentPropIndex := nCurrentPropIndex + 1;
refCmdData.n32Data[nCurrentPropIndex] := nOffsetLeftDrivingPin;
nCurrentPropIndex := nCurrentPropIndex + 1;
refCmdData.n32Data[nCurrentPropIndex] := nOffsetRightDrivingPin;
nCurrentPropIndex := nCurrentPropIndex + 1;
refCmdData.n32Data[nCurrentPropIndex] := nDrivingPinThickness;
nCurrentPropIndex := nCurrentPropIndex + 1;
refCmdData.n32Data[nCurrentPropIndex] := nTransferPosLeft;
nCurrentPropIndex := nCurrentPropIndex + 1;
refCmdData.n32Data[nCurrentPropIndex] := nTransferPosRight;
nCurrentPropIndex := nCurrentPropIndex + 1;
refCmdData.n32Data[nCurrentPropIndex] := nSafePosLeft;
nCurrentPropIndex := nCurrentPropIndex + 1;
refCmdData.n32Data[nCurrentPropIndex] := nSafePosRight;
nCurrentPropIndex := nCurrentPropIndex + 1;
refCmdData.n32Data[nCurrentPropIndex] := nTrayLength;
nCurrentPropIndex := nCurrentPropIndex + 1;
refCmdData.n32Data[nCurrentPropIndex] := nHollowDistance;
nCurrentPropIndex := nCurrentPropIndex + 1;
refCmdData.n32Data[nCurrentPropIndex] := nHollowWidth;
END_METHOD

METHOD M_GetSliderPosTrayInSlot : DINT
VAR_INPUT
	ePinSelection : E_DrivingPinSelection;
	eHollowSelection : E_TrayHollowSelection;
END_VAR
//Gibt die Position(Raw) für den Slider zurück, wenn Tray im Slot1 positioniert ist und entsprechender 
//DrivingPin in Mitte der ausgewählen Aussparung
CASE eHollowSelection OF
	E_TrayHollowSelection.Left:
		IF ePinSelection = E_DrivingPinSelection.Left THEN
			M_GetSliderPosTrayInSlot := REAL_TO_DINT(pTraySlot^.P_rRelPosX) + nHollowDistance + nOffsetLeftDrivingPin;
		ELSIF ePinSelection = E_DrivingPinSelection.Right THEN
			M_GetSliderPosTrayInSlot := REAL_TO_DINT(pTraySlot^.P_rRelPosX) + nHollowDistance - nOffsetRightDrivingPin;
		END_IF	
	E_TrayHollowSelection.Centre:
		IF ePinSelection = E_DrivingPinSelection.Left THEN
			M_GetSliderPosTrayInSlot := REAL_TO_DINT(pTraySlot^.P_rRelPosX) + nTrayLength / 2 + nOffsetLeftDrivingPin;
		ELSIF ePinSelection = E_DrivingPinSelection.Right THEN
			M_GetSliderPosTrayInSlot := REAL_TO_DINT(pTraySlot^.P_rRelPosX) + nTrayLength / 2 - nOffsetRightDrivingPin;
		END_IF	
	E_TrayHollowSelection.Right:
		IF ePinSelection = E_DrivingPinSelection.Left THEN
			M_GetSliderPosTrayInSlot := REAL_TO_DINT(pTraySlot^.P_rRelPosX) + nTrayLength - nHollowDistance + nOffsetLeftDrivingPin;
		ELSIF ePinSelection = E_DrivingPinSelection.Right THEN
			M_GetSliderPosTrayInSlot := REAL_TO_DINT(pTraySlot^.P_rRelPosX) + nTrayLength - nHollowDistance - nOffsetRightDrivingPin;
		END_IF
END_CASE
END_METHOD

METHOD M_GetSlot : POINTER TO FB_Slot
VAR_INPUT
	nSlotNr : UINT;
END_VAR
M_GetSlot := fbSlotList.M_GetAtNr(nSlotNr);
END_METHOD

METHOD M_GetSlotFromChild : POINTER TO FB_Slot
VAR_INPUT
	pObject : POINTER TO FB_Object;
END_VAR

VAR
	pSlot : POINTER TO FB_Slot;
END_VAR
//Die SlotList iterieren und vergleichen ob Objekte übereinstimmen
fbSlotList.M_SetCurrentToHead();
REPEAT
	pSlot := fbSlotList.M_GetNext();
	IF pSlot > 0 THEN
		IF pSlot^.P_pChild = pObject THEN
			M_GetSlotFromChild := pSlot;
			EXIT;
		END_IF
	END_IF
UNTIL pSlot = 0
END_REPEAT
END_METHOD

METHOD M_GetStateForTransfer : ERRORID
VAR_INPUT
	eCtrl : E_TransferTrayCtrl;
END_VAR
//Egal, welche Richtung was tranportiert wird, wenn Stacker, dann muss immer
//richtige Ausrichtung und auf einem Fach stehen
{IF defined(Stacker)}
IF afbStacker[1].P_eCurrentSpinPositon <> E_StackerRotPosition.TransferPositionPrinter1 THEN
	M_GetStateForTransfer := E_ErrorIdCmd.ERRORID_StackerNotInTransferPosition;
	RETURN;
END_IF
IF afbStacker[1].P_nCurrentShelf = 0 THEN
	M_GetStateForTransfer := E_ErrorIdCmd.ERRORID_StackerNotInShelfPosition;
	RETURN;
END_IF
{END_IF}

CASE eCtrl OF
	E_TransferTrayCtrl.LeftToSlot:
	{IF defined(Stacker)}
	IF afbStacker[1].P_bTraysAligned THEN
		IF afbStacker[1].P_bTrayInCurrentShelf THEN
			RETURN; //Alles OK
		ELSE
			M_GetStateForTransfer := E_ErrorIdCmd.ERRORID_NoTrayInStackerShelf;	
		END_IF
	ELSE
		M_GetStateForTransfer := E_ErrorIdCmd.ERRORID_TraysNotAligned;	
	END_IF
	{ELSE}
	IF NOT bReadyFlagLeft THEN
		M_GetStateForTransfer := E_ErrorIdCmd.ERRORID_NoTrayOnLeftTransferStation;
	END_IF
	{END_IF}
	E_TransferTrayCtrl.RightToSlot:
	{IF defined(Stacker)}
	IF afbStacker[1].P_bTraysAligned THEN
		IF afbStacker[1].P_bTrayInCurrentShelf THEN
			RETURN; //Alles OK
		ELSE
			M_GetStateForTransfer := E_ErrorIdCmd.ERRORID_NoTrayInStackerShelf;	
		END_IF
	ELSE
		M_GetStateForTransfer := E_ErrorIdCmd.ERRORID_TraysNotAligned;	
	END_IF
	{ELSE}
	IF NOT bReadyFlagRight THEN
		M_GetStateForTransfer := E_ErrorIdCmd.ERRORID_NoTrayOnRightTransferStation;
	END_IF
	{END_IF}
	E_TransferTrayCtrl.SlotToLeft:
	{IF defined(Stacker)}
	IF afbStacker[1].P_bTrayInCurrentShelf THEN
		M_GetStateForTransfer := E_ErrorIdCmd.ERRORID_TrayAlreadyInStackerShelf;
		RETURN;
	END_IF
	{ELSE}
	IF bReadyFlagLeft THEN
		M_GetStateForTransfer := E_ErrorIdCmd.ERRORID_TrayAlreadyOnLeftTransferStation;
	END_IF
	{END_IF}
	E_TransferTrayCtrl.SlotToRight:
	{IF defined(Stacker)}
	IF afbStacker[1].P_bTrayInCurrentShelf THEN
		M_GetStateForTransfer := E_ErrorIdCmd.ERRORID_TrayAlreadyInStackerShelf;
		RETURN;
	END_IF
	{ELSE}
	IF bReadyFlagRight THEN
		M_GetStateForTransfer := E_ErrorIdCmd.ERRORID_TrayAlreadyOnRightTransferStation;
	END_IF
	{END_IF}
ELSE
	M_GetStateForTransfer := E_ErrorIdCmd.ERRORID_InvalidCtrl;
END_CASE
END_METHOD

METHOD M_RemoveListEntry : BOOL
VAR_INPUT
	nSearchValue	: E_Action;
END_VAR
getPosPtr := 0;(* start from first node element *)
fbList.A_FindNext( hList := hList, putPosPtr := getPosPtr, putValue := nSearchValue, getValue=>getValue, getPosPtr=>getPosPtr );
IF fbList.bOk THEN	//Eintrag wurde gefunden
	fbList.A_RemoveValueAtPosPtr(hList:= hList,	putPosPtr:= getPosPtr);
	IF fbList.bOk THEN
		M_RemoveListEntry := TRUE;
	END_IF
END_IF
END_METHOD

METHOD M_SetAllProps : ERRORID
VAR_INPUT
	refCmdData : REFERENCE TO  ST_CmdData;
END_VAR

VAR
	i : UINT;
	pSlot 		: POINTER TO FB_Slot;
END_VAR
M_SetAllProps := SUPER^.M_SetAllProps(refCmdData);

IF M_SetAllProps > 0 THEN
	RETURN;
END_IF

{IF defined (TrayTransporterL)}
pSliderRef := ADR(fbHwRefTrayTransSlider);
pDrivingPinRefLeft := ADR(fbHwRefDrivingPinLeft);
pTrayLock := ADR(fbHwRefTrayLock);
{ELSIF defined (TrayTransporterR)}
pSliderRef := ADR(fbHwRefTrayTransSlider);
pDrivingPinRefRight := ADR(fbHwRefDrivingPinRight);
pTrayLock := ADR(fbHwRefTrayLock);
{ELSIF defined (TrayTransporterLR)}
pSliderRef := ADR(fbHwRefTrayTransSlider);
pDrivingPinRefLeft := ADR(fbHwRefDrivingPinLeft);
pDrivingPinRefRight := ADR(fbHwRefDrivingPinRight);
pTrayLock := ADR(fbHwRefTrayLock);
{ELSE}
M_SetAllProps := E_ErrorIdObjMgmt.ERRORID_InvalidHardwareRef;
RETURN;
{END_IF}

//Slots parametrieren
nCurrentPropIndex := nCurrentPropIndex + 1;
nFirstSlotPropIndex := nCurrentPropIndex;
nNumberOfSlots := DINT_TO_UINT(refCmdData.n32Data[nCurrentPropIndex]);

//Falls SlotList noch nicht existiert, dann neue erstellen
IF fbSlotList.P_nCount = 0 THEN
	FOR i:= 1 TO nNumberOfSlots BY 1 DO
		pSlot := __NEW(FB_Slot(pOwner := THIS));
		fbSlotList.M_Add(pSlot);
		nCurrentPropIndex := nCurrentPropIndex + 1;
		pSlot^.P_nNr := DINT_TO_USINT(refCmdData.n32Data[nCurrentPropIndex]);
		nCurrentPropIndex := nCurrentPropIndex + 1;
		pSlot^.P_rRelPosX := DINT_TO_REAL(refCmdData.n32Data[nCurrentPropIndex]);
		nCurrentPropIndex := nCurrentPropIndex + 1;
		pSlot^.P_rRelPosY := DINT_TO_REAL(refCmdData.n32Data[nCurrentPropIndex]);
		nCurrentPropIndex := nCurrentPropIndex + 1;
		pSlot^.P_rRelPosZ := DINT_TO_REAL(refCmdData.n32Data[nCurrentPropIndex]);
		IF i = 1 THEN
			pTraySlot := pSlot;
		END_IF
	END_FOR
ELSE
	IF nNumberOfSlots <> fbSlotList.P_nCount THEN	//Anzahl der Slots dürfen sich nicht ändern
		M_SetAllProps := E_ErrorIdObjMgmt.ERRORID_ChangeNoOfSlotsNotAllowed;
		RETURN;		
	END_IF

	FOR i:= 1 TO nNumberOfSlots BY 1 DO
		nCurrentPropIndex := nCurrentPropIndex + 1;
		pSlot := fbSlotList.M_GetAtNr(DINT_TO_USINT(refCmdData.n32Data[nCurrentPropIndex]));
		IF pSlot > 0 THEN
			nCurrentPropIndex := nCurrentPropIndex + 1;
			pSlot^.P_rRelPosX := DINT_TO_REAL(refCmdData.n32Data[nCurrentPropIndex]);
			nCurrentPropIndex := nCurrentPropIndex + 1;
			pSlot^.P_rRelPosY := DINT_TO_REAL(refCmdData.n32Data[nCurrentPropIndex]);
			nCurrentPropIndex := nCurrentPropIndex + 1;
			pSlot^.P_rRelPosZ := DINT_TO_REAL(refCmdData.n32Data[nCurrentPropIndex]);
		ELSE
			M_SetAllProps := 222;
			RETURN;
		END_IF	
	END_FOR
END_IF
nLastSlotPropIndex := nCurrentPropIndex;

nCurrentPropIndex := nCurrentPropIndex + 1;
nSpecPropIndex := nCurrentPropIndex;

nOffsetLeftDrivingPin := refCmdData.n32Data[nCurrentPropIndex];
nCurrentPropIndex := nCurrentPropIndex + 1;
nOffsetRightDrivingPin := refCmdData.n32Data[nCurrentPropIndex];
nCurrentPropIndex := nCurrentPropIndex + 1;
nDrivingPinThickness := refCmdData.n32Data[nCurrentPropIndex];
nCurrentPropIndex := nCurrentPropIndex + 1;
nTransferPosLeft := refCmdData.n32Data[nCurrentPropIndex];
nCurrentPropIndex := nCurrentPropIndex + 1;
nTransferPosRight := refCmdData.n32Data[nCurrentPropIndex];
nCurrentPropIndex := nCurrentPropIndex + 1;
nSafePosLeft := refCmdData.n32Data[nCurrentPropIndex];
nCurrentPropIndex := nCurrentPropIndex + 1;
nSafePosRight := refCmdData.n32Data[nCurrentPropIndex];
nCurrentPropIndex := nCurrentPropIndex + 1;
nTrayLength := refCmdData.n32Data[nCurrentPropIndex];
nCurrentPropIndex := nCurrentPropIndex + 1;
nHollowDistance := refCmdData.n32Data[nCurrentPropIndex];
nCurrentPropIndex := nCurrentPropIndex + 1;
nHollowWidth := refCmdData.n32Data[nCurrentPropIndex];

nNoOfProps := nCurrentPropIndex + 1;
END_METHOD

METHOD M_SetSingleProp : ERRORID
VAR_INPUT
	refCmdData : REFERENCE TO  ST_CmdData;
END_VAR
IF nSpecPropIndex = refCmdData.aHeader[1] THEN
	nOffsetLeftDrivingPin := refCmdData.n32Data[0];
ELSIF (nSpecPropIndex + 1) = refCmdData.aHeader[1] THEN
	nOffsetRightDrivingPin := refCmdData.n32Data[0];
ELSIF (nSpecPropIndex + 2) = refCmdData.aHeader[1] THEN
	nDrivingPinThickness := refCmdData.n32Data[0];
ELSIF (nSpecPropIndex + 3) = refCmdData.aHeader[1] THEN
	nTransferPosLeft := refCmdData.n32Data[0];
ELSIF (nSpecPropIndex + 4) = refCmdData.aHeader[1] THEN
	nTransferPosRight := refCmdData.n32Data[0];
ELSIF (nSpecPropIndex + 5) = refCmdData.aHeader[1] THEN
	nSafePosLeft := refCmdData.n32Data[0];
ELSIF (nSpecPropIndex + 6) = refCmdData.aHeader[1] THEN
	nSafePosRight := refCmdData.n32Data[0];
ELSIF (nSpecPropIndex + 7) = refCmdData.aHeader[1] THEN
	nTrayLength := refCmdData.n32Data[0];
ELSIF (nSpecPropIndex + 8) = refCmdData.aHeader[1] THEN
	nHollowDistance := refCmdData.n32Data[0];
ELSIF (nSpecPropIndex + 9) = refCmdData.aHeader[1] THEN
	nHollowWidth := refCmdData.n32Data[0];	
ELSE
	M_SetSingleProp := SUPER^.M_SetSingleProp(refCmdData);
END_IF
END_METHOD

METHOD M_Stop : ERRORID
IF bInit OR bMoveSlider OR bTurnDrivingPin THEN
	bStop := TRUE;	
END_IF
END_METHOD

PROPERTY P_bReadyForDeliveringLeft : BOOL
GET
{IF defined(Stacker)}
//Stacker muss auf TransferPosPrinter1 stehen
//Stacker muss auf irgendeinem Shelf stehen
//Trays müssen hier nicht unbedingt ausgerichtet sein?
//Sensor "TrayDetection" muss FALSE sein
P_bReadyForDeliveringLeft := (afbStacker[1].P_eCurrentSpinPositon = E_StackerRotPosition.TransferPositionPrinter1) AND
 						(afbStacker[1].P_nCurrentShelf > 0) AND afbStacker[1].P_bTraysAligned AND NOT afbStacker[1].P_bTrayInCurrentShelf;
{ELSE}
P_bReadyForDeliveringLeft := NOT bReadyFlagLeft;
{END_IF}
END_GET
END_PROPERTY

PROPERTY P_bReadyForDeliveringRight : BOOL
GET
P_bReadyForDeliveringRight := NOT bReadyFlagRight;
END_GET
END_PROPERTY

PROPERTY P_bReadyForTakingLeft : BOOL
GET
{IF defined(Stacker)}
//Stacker muss auf TransferPosPrinter1 stehen
//Stacker muss auf irgendeinem Shelf stehen
//Trays müssen genau ausgerichtet sein (Aligned)
//Sensor "TrayDetection" muss TRUE sein
P_bReadyForTakingLeft := (afbStacker[1].P_eCurrentSpinPositon = E_StackerRotPosition.TransferPositionPrinter1) AND
 						(afbStacker[1].P_nCurrentShelf > 0) AND afbStacker[1].P_bTraysAligned AND (afbStacker[1].P_bTrayInCurrentShelf);
{ELSE}
P_bReadyForTakingLeft := bReadyFlagLeft;
{END_IF}
END_GET
END_PROPERTY

PROPERTY P_bReadyForTakingRight : BOOL
GET
P_bReadyForTakingRight := bReadyFlagRight;
END_GET
END_PROPERTY

PROPERTY P_bStopAllOnError : BOOL
GET
END_GET
END_PROPERTY

PROPERTY P_nDrivingPinGap : DINT
GET
P_nDrivingPinGap := (nHollowWidth - nDrivingPinThickness) / 2;
END_GET
END_PROPERTY

PROPERTY P_nHollowDistance : DINT
GET
P_nHollowDistance := nHollowDistance;
END_GET
END_PROPERTY

PROPERTY P_nHollowToHollow : DINT
GET
P_nHollowToHollow := nTrayLength - 2 * nHollowDistance;
END_GET
END_PROPERTY

PROPERTY P_nMaxSliderPos : DINT
GET
P_nMaxSliderPos := pSliderRef^.P_nMaxPos;
END_GET
END_PROPERTY

PROPERTY P_nMaxSliderSpeed : DINT
GET
P_nMaxSliderSpeed := pSliderRef^.P_nMaxSpeed;
END_GET
END_PROPERTY

PROPERTY P_nMinSliderPos : DINT
GET
P_nMinSliderPos := pSliderRef^.P_nMinPos;
END_GET
END_PROPERTY

PROPERTY P_nSafePosLeft : DINT
GET
P_nSafePosLeft := nSafePosLeft;
END_GET
END_PROPERTY

PROPERTY P_nSafePosRight : DINT
GET
P_nSafePosRight := nSafePosRight;
END_GET
END_PROPERTY

PROPERTY P_nTransferPosLeft : DINT
GET
P_nTransferPosLeft := nTransferPosLeft;
END_GET
END_PROPERTY

PROPERTY P_nTransferPosRight : DINT
GET
P_nTransferPosRight := nTransferPosRight;
END_GET
END_PROPERTY

PROPERTY P_nTrayLength : DINT
GET
P_nTrayLength := nTrayLength;
END_GET
END_PROPERTY

END_FUNCTION_BLOCK

// ---- Hardware/NanotecPanDrive/FB_HwRefNanotecPD.TcPOU
FUNCTION_BLOCK FB_HwRefNanotecPD EXTENDS FB_CanNodeBase
VAR_INPUT
	nControlword	AT%Q* : UINT;
	nMode			AT%Q* : SINT;
	nTargetPosition AT%Q* : DINT;
	nTargetSpeed	AT%Q* : INT;
	nDriveSubMode	AT%Q* : UDINT; //1 für Move, 8 für Stillstand mit Stromabsenkung	
END_VAR
VAR_OUTPUT
	nStatusword 	 	AT%I* : UINT;
	nCurrentMode 	 	AT%I* : SINT;
	nCurrentPosition 	AT%I* : DINT;
	nCurrentSpeed		AT%I* : INT;
	nFollowingError		AT%I* : DINT;	
END_VAR
VAR
	bIsHomed 				: BOOL;
	eCurrentSTM				: E_CoDS402States;
	nState 					: USINT;
	bFirstTimeInOperational : BOOL := TRUE;
	
	nStateA_ProcessError	: USINT;
	nLastErrorID			: DWORD;
	nErrorCount				: USINT;
	
	nStateA_ResetError		: USINT;
END_VAR

VAR PERSISTENT
	nDistPerMotorRev	: DINT;
	nRefPos				: DINT;
	nHomePos			: DINT;
	nSlowHomingSpeed	: DINT;
	nFastHomingSpeed	: DINT;
	bInvertInitDir		: BOOL;
	nMinPos				: DINT;
	nMaxPos				: DINT;
	nMaxSpeed			: DINT;
END_VAR

//In der Basisklasse wird A_Prepare und A_ResetApp ausgeführt
//ResetApp ist hier nicht relevant.

eCurrentSTM := M_GetDS402State();
CASE nState OF
	0:	//Prepare
		SUPER^();
		IF bPreparingOK THEN
			nState := 1;
		END_IF
		
	1:	//Operational
		//Wenn hier zum erstem mal hineingesprungen wird, und in error, dann gleich resetten
		IF eCurrentSTM = E_CoDS402States.DS402STATE_Fault OR eCurrentSTM = E_CoDS402States.DS402STATE_FaultReactionActive THEN
			IF bFirstTimeInOperational THEN
				nState := 4;
			ELSE
				nState := 2;
			END_IF
		END_IF
		bFirstTimeInOperational := FALSE;
		
	2:	//Process error
		A_ProcessError();
		IF nStateA_ProcessError = 80 THEN
			//Error auswerten - es werden nur die untersten 16Bit ausgewertet (Error Code siehe Doku NanoTec)
			nLastErrorID := nLastErrorID AND 16#FFFF;
			CASE nLastErrorID OF
				16#1000:	nErrorID := E_ErrorIdHwGeneral.ERRORID_GenericError;
				16#2300:	nErrorID := E_ErrorIdHwGeneral.ERRORID_MotorCurrentExceeded;
				16#3100:	nErrorID := E_ErrorIdHwGeneral.ERRORID_InvalidInputVoltage;
				16#4200:	nErrorID := E_ErrorIdHwGeneral.ERRORID_ControllerTemperature;
				16#5540:	nErrorID := E_ErrorIdHwGeneral.ERRORID_InterlockError;
				16#6010:	nErrorID := E_ErrorIdHwGeneral.ERRORID_SoftwareReset;
				16#6100:	nErrorID := E_ErrorIdHwGeneral.ERRORID_InternalSoftwareError;
				16#6320:	nErrorID := E_ErrorIdHwGeneral.ERRORID_InvalidRatedCurrent;
				16#7113:	nErrorID := E_ErrorIdHwGeneral.ERRORID_BallastResistorOverloaded;
				16#7121:	nErrorID := E_ErrorIdHwGeneral.ERRORID_MotorBlocked;
				16#7200:	nErrorID := E_ErrorIdHwGeneral.ERRORID_InternalError;
				16#7305:	nErrorID := E_ErrorIdHwGeneral.ERRORID_Sensor1Fault;
				16#7306:	nErrorID := E_ErrorIdHwGeneral.ERRORID_Sensor2Fault;
				16#7307:	nErrorID := E_ErrorIdHwGeneral.ERRORID_SensorNFault;
				16#7600:	nErrorID := E_ErrorIdHwGeneral.ERRORID_MemoryError;
				16#8000,16#8100: nErrorID := E_ErrorIdHwGeneral.ERRORID_FieldbusMonitoring;
				16#8130, 16#8200, 16#8210, 16#8220, 16#8240 : nErrorID := E_ErrorIdHwGeneral.ERRORID_CANopenError;	
				16#8400:	nErrorID := E_ErrorIdHwGeneral.ERRORID_SpeedMonitoring;
				16#8611:	nErrorID := E_ErrorIdHwGeneral.ERRORID_FollowingError;
				16#8612:	nErrorID := E_ErrorIdHwGeneral.ERRORID_LimitSwitchExceeded;
			ELSE
				nErrorID := 0;
			END_CASE
			nStateA_ProcessError := 0;
			//Notify error
			stError.HardwareGrp := stHardwareId.eGroup;
			stError.HardwareNr := stHardwareId.nItem;
			stError.POU := E_POU.POU_FB_HwRefNanotecPD;
			stError.POUAction := E_POUACT.POUACT_UNDEFIEND;
			stError.ErrorId := nErrorID;
			fbErrorList.M_Add(stError);
			nState := 3;
		END_IF
		
	3:	//Error
		IF bResetError THEN
			nState:= 4;
			bResetError := FALSE;
		END_IF
		bIsHomed := FALSE;
		bError := TRUE;
		
	4:	//Reset
		bBusy := TRUE;
		A_ResetError();
		IF nStateA_ResetError = 80 THEN
			bError := FALSE;
			bBusy := FALSE;
			nStateA_ResetError := 0;
			nState := 1;
		ELSIF nStateA_ResetError = 99 THEN
			bBusy := FALSE;
			nStateA_ResetError := 0;
			nState := 3;
		END_IF
	
END_CASE

ACTION A_ProcessError:
IF nStateA_ProcessError = 0 THEN
	//Object 0x1003:00 auslesen (Anzahl der Errors im Pre-defined error field)
	fbSdoRead(nIndex:= 16#1003, nSubIndex:= 0, nDataLength:= 1, bExecute:= TRUE);
	nErrorCount := 0;
	IF NOT fbSdoRead.bBusy THEN
		IF NOT fbSdoRead.bError THEN
			nErrorCount := DINT_TO_USINT(fbSdoRead.nData);
		END_IF
		fbSdoRead(bExecute:= FALSE);
		IF nErrorCount > 0 THEN
			nStateA_ProcessError := 1;
		ELSE
			nStateA_ProcessError := 80;
		END_IF
	END_IF
END_IF


IF nStateA_ProcessError = 1 THEN
	//Object 0x1003:01 auslesen (Neuester Error)
	fbSdoRead(nIndex:= 16#1003, nSubIndex:= 1, nDataLength:= 4, bExecute:= TRUE);
	nLastErrorID := 0;
	IF NOT fbSdoRead.bBusy THEN
		IF NOT fbSdoRead.bError THEN
			nLastErrorID := fbSdoRead.nData;
		END_IF
		fbSdoRead(bExecute:= FALSE);
		nStateA_ProcessError := 80;
	END_IF
END_IF
END_ACTION

ACTION A_ResetError:
CASE nStateA_ResetError OF
	0:	
		CASE eCurrentSTM OF
			E_CoDS402States.DS402STATE_Fault:
				nControlword := 153;	//Reset error
			E_CoDS402States.DS402STATE_SwitchOnDisabled:
				nStateA_ResetError := 1;
			E_CoDS402States.DS402STATE_ReadyToSwitchOn:
				nControlword := 0;	//Transition 7 in DS402 statemachine -> geht in Switch on disabled
				nStateA_ResetError := 1;
			E_CoDS402States.DS402STATE_SwitchedOn:
				nControlword := 0;	//Transition 10 in DS402 statemachine -> geht in Switch on disabled
				nStateA_ResetError := 1;
			E_CoDS402States.DS402STATE_OperationEnabled:
				nControlword := 0;	//Shutdown
				nStateA_ResetError := 1;
			E_CoDS402States.DS402STATE_NotReadyToSwitchOn:	//Statusword wahrscheinlich nicht gemappt
				nStateA_ResetError := 99;
		END_CASE
		
	1:	//Würde Antrieb bereits gehomed?
		IF bIsHomed THEN
			nControlword := 6;
			nStateA_ResetError := 2;
		ELSE
			nStateA_ResetError := 80;
		END_IF
		
	2:	IF eCurrentSTM = E_CoDS402States.DS402STATE_ReadyToSwitchOn THEN
			nControlword := 7;	//Change to "Switched on"
			nStateA_ResetError := 3;
		ELSIF eCurrentSTM = E_CoDS402States.DS402STATE_Fault THEN
			nStateA_ResetError := 99;
		END_IF
	
	3:	IF eCurrentSTM = E_CoDS402States.DS402STATE_SwitchedOn THEN
			nControlword := 15;	//Change to "Switched on"
			nStateA_ResetError := 4;
		ELSIF eCurrentSTM = E_CoDS402States.DS402STATE_Fault THEN
			nStateA_ResetError := 99;
		END_IF
		
	4:	IF eCurrentSTM = E_CoDS402States.DS402STATE_OperationEnabled THEN
			nStateA_ResetError := 80;
		ELSIF eCurrentSTM = E_CoDS402States.DS402STATE_Fault THEN
			nStateA_ResetError := 99;
		END_IF		
	
END_CASE
END_ACTION

METHOD M_GetDS402State : E_CoDS402States
VAR_INPUT
END_VAR
IF (nStatusword AND 16#4F) = 0 THEN
	M_GetDS402State := E_CoDS402States.DS402STATE_NotReadyToSwitchOn;
ELSIF (nStatusword AND 16#4F) = 16#40 THEN
	M_GetDS402State := E_CoDS402States.DS402STATE_SwitchOnDisabled;
ELSIF (nStatusword AND 16#6F) = 16#21 THEN
	M_GetDS402State := E_CoDS402States.DS402STATE_ReadyToSwitchOn;
ELSIF (nStatusword AND 16#6F) = 16#23 THEN
	M_GetDS402State := E_CoDS402States.DS402STATE_SwitchedOn;
ELSIF (nStatusword AND 16#6F) = 16#27 THEN
	M_GetDS402State := E_CoDS402States.DS402STATE_OperationEnabled;
ELSIF (nStatusword AND 16#6F) = 16#07 THEN
	M_GetDS402State := E_CoDS402States.DS402STATE_QuickStopActive;
ELSIF (nStatusword AND 16#4F) = 16#0F THEN
	M_GetDS402State := E_CoDS402States.DS402STATE_FaultReactionActive;
ELSIF (nStatusword AND 16#4F) = 16#08 THEN
	M_GetDS402State := E_CoDS402States.DS402STATE_Fault;
ELSE
	M_GetDS402State := E_CoDS402States.DS402STATE_Notspecified;
END_IF
END_METHOD

METHOD M_GetHomingState : E_CoDS402HomingState
VAR_INPUT
END_VAR

VAR 
END_VAR
//werted nur die Bits 10,12,13 vom Statusword aus
CASE nStatusword AND 16#3400 OF
	16#0000:	M_GetHomingState := E_CoDS402HomingState.HomingInProgress;
	16#0400:	M_GetHomingState := E_CoDS402HomingState.HomingInteruptedOrNotReached;
	16#1000:	M_GetHomingState := E_CoDS402HomingState.HomingAttainedButNotReached;
	16#1400:	M_GetHomingState := E_CoDS402HomingState.HomingSuccess;
	16#2000,
	16#2400		:M_GetHomingState := E_CoDS402HomingState.HomingError;
END_CASE
END_METHOD

METHOD M_RealToInternPos : DINT
VAR_INPUT
	nValue : DINT;
END_VAR
M_RealToInternPos := REAL_TO_DINT(DINT_TO_REAL(nValue) * 2000.0 / DINT_TO_REAL(nDistPerMotorRev));
END_METHOD

METHOD M_RealToInternSpeed : INT
VAR_INPUT
	nValue : DINT; //Speed in µm/s oder 1/100°/sec
END_VAR
//Umrechnung in U/min
M_RealToInternSpeed := REAL_TO_INT(DINT_TO_REAL(nValue) / DINT_TO_REAL(nDistPerMotorRev) * 60.0);
RETURN;
END_METHOD

METHOD M_SetTargetPos : BOOL
VAR_INPUT
	nValue : DINT; //Reale Einheit
END_VAR
IF (nValue >= nMinPos) AND (nValue <= nMaxPos) THEN
	nTargetPosition :=  REAL_TO_DINT(DINT_TO_REAL(nValue) * 2000.0 / DINT_TO_REAL(nDistPerMotorRev));
	M_SetTargetPos := TRUE;
END_IF
END_METHOD

METHOD M_SetTargetSpeed : BOOL
VAR_INPUT
	nValue : DINT; //Reale Einheit
END_VAR
IF (nValue >= 0) AND (nValue <= nMaxSpeed) THEN
	nTargetSpeed := M_RealToInternSpeed(nValue);
	M_SetTargetSpeed := TRUE;
END_IF
END_METHOD

PROPERTY P_bInvertInitDir : BOOL
GET
P_bInvertInitDir := bInvertInitDir;
END_GET
SET
bInvertInitDir := P_bInvertInitDir;
fbSettings.M_WritePersData();
END_SET
END_PROPERTY

PROPERTY P_bIsHomed : BOOL
GET
P_bIsHomed := bIsHomed;
END_GET
SET
bIsHomed := P_bIsHomed;
END_SET
END_PROPERTY

PROPERTY P_nCurrentRealPos : DINT
GET
P_nCurrentRealPos := REAL_TO_DINT(DINT_TO_REAL(nCurrentPosition) / 2000.0 * DINT_TO_REAL(nDistPerMotorRev));
END_GET
END_PROPERTY

PROPERTY P_nDistPerMotorRev : DINT
GET
P_nDistPerMotorRev := nDistPerMotorRev;
END_GET
SET
nDistPerMotorRev := P_nDistPerMotorRev;
fbSettings.M_WritePersData();
END_SET
END_PROPERTY

PROPERTY P_nErrorID : ERRORID
GET
P_nErrorID := nErrorId;
END_GET
END_PROPERTY

PROPERTY P_nFastHomingSpeed : DINT
GET
P_nFastHomingSpeed := nFastHomingSpeed;
END_GET
SET
nFastHomingSpeed := P_nFastHomingSpeed;
fbSettings.M_WritePersData();
END_SET
END_PROPERTY

PROPERTY P_nHomePos : DINT
GET
P_nHomePos := nHomePos;
END_GET
SET
nHomePos := P_nHomePos;
fbSettings.M_WritePersData();
END_SET
END_PROPERTY

PROPERTY P_nMaxPos : DINT
GET
P_nMaxPos := nMaxPos;
END_GET
SET
nMaxPos := P_nMaxPos;
fbSettings.M_WritePersData();
END_SET
END_PROPERTY

PROPERTY P_nMaxSpeed : DINT
GET
P_nMaxSpeed := nMaxSpeed;
END_GET
SET
nMaxSpeed := P_nMaxSpeed;
fbSettings.M_WritePersData();
END_SET
END_PROPERTY

PROPERTY P_nMinPos : DINT
GET
P_nMinPos := nMinPos;
END_GET
SET
nMinPos := P_nMinPos;
fbSettings.M_WritePersData();
END_SET
END_PROPERTY

PROPERTY P_nRefPos : DINT
GET
P_nRefPos := nRefPos;
END_GET
SET
nRefPos := P_nRefPos;
fbSettings.M_WritePersData();
END_SET
END_PROPERTY

PROPERTY P_nSlowHomingSpeed : DINT
GET
P_nSlowHomingSpeed := nSlowHomingSpeed;
END_GET
SET
nSlowHomingSpeed := P_nSlowHomingSpeed;
fbSettings.M_WritePersData();
END_SET
END_PROPERTY

END_FUNCTION_BLOCK

// ---- Hardware/TrayLock/FB_HwRefTrayLock.TcPOU
FUNCTION_BLOCK FB_HwRefTrayLock
VAR_INPUT
	bLock  			AT %Q* : BOOL;
	bUnlock  		AT %Q* : BOOL;
	bDisableHeater 	AT %Q* : BOOL;
END_VAR
VAR_OUTPUT
	bLocked			AT %I* : BOOL;
	bUnlocked		AT %I* : BOOL;
	eCurrentState : E_LockState;
END_VAR
VAR
END_VAR

IF bLocked THEN
	eCurrentState := E_LockState.Locked;
ELSIF bUnlocked THEN
	eCurrentState := E_LockState.Unlocked;
ELSE
	eCurrentState := E_LockState.UNDEFINIED;
END_IF

PROPERTY P_bFeedback : BOOL
GET
P_bFeedback := F_GetMappingStatus(ADR(bLocked), SIZEOF(bLocked)) = EPlcMappingStatus.MS_Partial AND 
				F_GetMappingStatus(ADR(bUnlocked), SIZEOF(bUnlocked)) = EPlcMappingStatus.MS_Partial;
END_GET
END_PROPERTY

END_FUNCTION_BLOCK

// ---- Hardware/NanotecPanDrive/FB_NanotecPD_Power.TcPOU
FUNCTION_BLOCK FB_NanotecPD_Power
VAR_INPUT
	bExecute : BOOL;
END_VAR
VAR_OUTPUT
	bBusy 		: BOOL;
	bError 		: BOOL;
	nErrorId 	: ERRORID;	
END_VAR
VAR_IN_OUT
	pHwRef : POINTER TO FB_HwRefNanotecPD; 
END_VAR
VAR
	nState : USINT;
	fbSdoWrite : FB_SDO_WRITE;
END_VAR

//Achtung, anders als bei TMCM-Controllern wird die Statemachine des Controller hier nur bis "SwitchedOn" durchlaufen.
//"OperationEnabled" wird erst nach dem Setzen des Modes gesetzt. Jedes Ändern des Modes erfordert eine Rückkehr zu "SwitchedOn"
IF bExecute THEN
	IF nState = 0 THEN
		bBusy := TRUE;
		CASE pHwRef^.M_GetDS402State() OF
			E_CoDS402States.DS402STATE_Fault:
				pHwRef^.nControlword := 153;	//Reset Error
			E_CoDS402States.DS402STATE_SwitchOnDisabled:
				nState := 1;
			E_CoDS402States.DS402STATE_ReadyToSwitchOn:
				pHwRef^.nControlword := 0;	//Transition 7 in DS402 statemachine -> geht in Switch on disabled
				nState := 1;
			E_CoDS402States.DS402STATE_SwitchedOn:
				pHwRef^.nControlword := 0;	//Transition 10 in DS402 statemachine -> geht in Switch on disabled
				nState := 1;
			E_CoDS402States.DS402STATE_OperationEnabled:
				pHwRef^.nControlword := 0;	//Shutdown
				nState := 1;
			E_CoDS402States.DS402STATE_NotReadyToSwitchOn:
				nErrorId := E_ErrorIdDS402.ERRORID_NotReadyToSwitchOn;
				nState := 99;
		END_CASE
 	END_IF
	
	CASE nState OF
		1:	//Change ro "Ready to switched on"
			pHwRef^.nControlword := 6;
			nState := 2;
			
		2:	//State = "Ready to switched on" ? -> Switch on
			IF pHwRef^.M_GetDS402State() = E_CoDS402States.DS402STATE_ReadyToSwitchOn THEN
				pHwRef^.nControlword := 7;
				nState := 3;
			ELSIF pHwRef^.M_GetDS402State() = E_CoDS402States.DS402STATE_Fault THEN
				nErrorId := E_ErrorIdDS402.ERRORID_FaultState;
				nState := 99;
			END_IF
			
		3:	//State = "Switched on" ?
			IF pHwRef^.M_GetDS402State() = E_CoDS402States.DS402STATE_SwitchedOn THEN
				//pHwRef^.nDriveSubMode := 1;
				nState := 80;
			ELSIF pHwRef^.M_GetDS402State() = E_CoDS402States.DS402STATE_Fault THEN
				nErrorId := E_ErrorIdDS402.ERRORID_FaultState;
				nState := 99;
			END_IF
			
	END_CASE
	
	IF nState >= 80 THEN
		bBusy := FALSE;
		IF nState = 99 THEN
			bError := TRUE;
		END_IF
	END_IF
	
ELSE
	bError := FALSE;
	nErrorId := 0;
	nState := 0;
END_IF

END_FUNCTION_BLOCK

